LIN {X -289.657,Y 14.097,Z 88.630,A -2.786,B 90.000,C 0.000} C_DIS
LIN {X -289.655,Y 14.148,Z 88.567,A -2.796,B 90.000,C 0.000} C_DIS
LIN {X -289.652,Y 14.199,Z 88.524,A -2.806,B 90.000,C 0.000} C_DIS
LIN {X -289.650,Y 14.241,Z 88.320,A -2.815,B 90.000,C 0.000} C_DIS
LIN {X -289.648,Y 14.292,Z 88.278,A -2.825,B 90.000,C 0.000} C_DIS
LIN {X -289.645,Y 14.343,Z 88.214,A -2.835,B 90.000,C 0.000} C_DIS
LIN {X -289.643,Y 14.385,Z 87.908,A -2.843,B 90.000,C 0.000} C_DIS
LIN {X -289.640,Y 14.436,Z 87.844,A -2.853,B 90.000,C 0.000} C_DIS
LIN {X -289.638,Y 14.487,Z 87.801,A -2.863,B 90.000,C 0.000} C_DIS
LIN {X -289.636,Y 14.530,Z 87.597,A -2.872,B 90.000,C 0.000} C_DIS
LIN {X -289.633,Y 14.581,Z 87.555,A -2.882,B 90.000,C 0.000} C_DIS
LIN {X -289.631,Y 14.632,Z 87.491,A -2.892,B 90.000,C 0.000} C_DIS
LIN {X -289.629,Y 14.674,Z 87.185,A -2.900,B 90.000,C 0.000} C_DIS
LIN {X -289.626,Y 14.725,Z 87.121,A -2.910,B 90.000,C 0.000} C_DIS
LIN {X -289.623,Y 14.776,Z 87.079,A -2.921,B 90.000,C 0.000} C_DIS
LIN {X -289.621,Y 14.818,Z 86.875,A -2.929,B 90.000,C 0.000} C_DIS
LIN {X -289.619,Y 14.869,Z 86.832,A -2.939,B 90.000,C 0.000} C_DIS
LIN {X -289.616,Y 14.920,Z 86.769,A -2.949,B 90.000,C 0.000} C_DIS
LIN {X -289.614,Y 14.963,Z 86.462,A -2.958,B 90.000,C 0.000} C_DIS
LIN {X -289.611,Y 15.014,Z 86.399,A -2.968,B 90.000,C 0.000} C_DIS
LIN {X -289.608,Y 15.065,Z 86.356,A -2.978,B 90.000,C 0.000} C_DIS
LIN {X -289.606,Y 15.107,Z 86.152,A -2.986,B 90.000,C 0.000} C_DIS
LIN {X -289.604,Y 15.158,Z 86.110,A -2.996,B 90.000,C 0.000} C_DIS
LIN {X -289.601,Y 15.209,Z 86.046,A -3.006,B 90.000,C 0.000} C_DIS
LIN {X -289.599,Y 15.251,Z 85.740,A -3.015,B 90.000,C 0.000} C_DIS
LIN {X -289.596,Y 15.302,Z 85.676,A -3.025,B 90.000,C 0.000} C_DIS
LIN {X -289.593,Y 15.353,Z 85.634,A -3.035,B 90.000,C 0.000} C_DIS
LIN {X -289.591,Y 15.396,Z 85.429,A -3.043,B 90.000,C 0.000} C_DIS
LIN {X -289.588,Y 15.447,Z 85.387,A -3.053,B 90.000,C 0.000} C_DIS
LIN {X -289.586,Y 15.498,Z 85.323,A -3.063,B 90.000,C 0.000} C_DIS
LIN {X -289.583,Y 15.540,Z 85.017,A -3.072,B 90.000,C 0.000} C_DIS
LIN {X -289.578,Y 15.642,Z 84.890,A -3.092,B 90.000,C 0.000} C_DIS
LIN {X -289.576,Y 15.684,Z 84.583,A -3.100,B 90.000,C 0.000} C_DIS
LIN {X -289.573,Y 15.735,Z 84.520,A -3.110,B 90.000,C 0.000} C_DIS
LIN {X -289.570,Y 15.786,Z 84.477,A -3.120,B 90.000,C 0.000} C_DIS
LIN {X -289.568,Y 15.829,Z 84.273,A -3.129,B 90.000,C 0.000} C_DIS
LIN {X -289.565,Y 15.880,Z 84.231,A -3.139,B 90.000,C 0.000} C_DIS
LIN {X -289.562,Y 15.931,Z 84.167,A -3.149,B 90.000,C 0.000} C_DIS
LIN {X -289.560,Y 15.973,Z 83.861,A -3.157,B 90.000,C 0.000} C_DIS
LIN {X -289.557,Y 16.024,Z 83.797,A -3.167,B 90.000,C 0.000} C_DIS
LIN {X -289.554,Y 16.075,Z 83.755,A -3.178,B 90.000,C 0.000} C_DIS
LIN {X -289.552,Y 16.117,Z 83.551,A -3.186,B 90.000,C 0.000} C_DIS
LIN {X -289.549,Y 16.168,Z 83.508,A -3.196,B 90.000,C 0.000} C_DIS
LIN {X -289.546,Y 16.219,Z 83.444,A -3.206,B 90.000,C 0.000} C_DIS
LIN {X -289.544,Y 16.262,Z 83.138,A -3.214,B 90.000,C 0.000} C_DIS
LIN {X -289.541,Y 16.312,Z 83.075,A -3.225,B 90.000,C 0.000} C_DIS
LIN {X -289.538,Y 16.363,Z 83.032,A -3.235,B 90.000,C 0.000} C_DIS
LIN {X -289.536,Y 16.406,Z 82.828,A -3.243,B 90.000,C 0.000} C_DIS
LIN {X -289.533,Y 16.457,Z 82.785,A -3.253,B 90.000,C 0.000} C_DIS
LIN {X -289.530,Y 16.508,Z 82.722,A -3.263,B 90.000,C 0.000} C_DIS
LIN {X -289.527,Y 16.550,Z 82.416,A -3.272,B 90.000,C 0.000} C_DIS
LIN {X -289.524,Y 16.601,Z 82.352,A -3.282,B 90.000,C 0.000} C_DIS
LIN {X -289.522,Y 16.652,Z 82.309,A -3.292,B 90.000,C 0.000} C_DIS
LIN {X -289.519,Y 16.694,Z 82.105,A -3.300,B 90.000,C 0.000} C_DIS
LIN {X -289.516,Y 16.745,Z 82.063,A -3.310,B 90.000,C 0.000} C_DIS
LIN {X -289.513,Y 16.796,Z 81.999,A -3.320,B 90.000,C 0.000} C_DIS
LIN {X -289.511,Y 16.839,Z 81.693,A -3.329,B 90.000,C 0.000} C_DIS
LIN {X -289.508,Y 16.890,Z 81.629,A -3.339,B 90.000,C 0.000} C_DIS
LIN {X -289.505,Y 16.941,Z 81.587,A -3.349,B 90.000,C 0.000} C_DIS
LIN {X -289.502,Y 16.983,Z 81.383,A -3.357,B 90.000,C 0.000} C_DIS
LIN {X -289.499,Y 17.034,Z 81.340,A -3.367,B 90.000,C 0.000} C_DIS
LIN {X -289.496,Y 17.085,Z 81.276,A -3.377,B 90.000,C 0.000} C_DIS
LIN {X -289.494,Y 17.127,Z 80.970,A -3.386,B 90.000,C 0.000} C_DIS
LIN {X -289.491,Y 17.178,Z 80.907,A -3.396,B 90.000,C 0.000} C_DIS
LIN {X -289.488,Y 17.229,Z 80.864,A -3.406,B 90.000,C 0.000} C_DIS
LIN {X -289.485,Y 17.272,Z 80.660,A -3.414,B 90.000,C 0.000} C_DIS
LIN {X -289.482,Y 17.322,Z 80.618,A -3.424,B 90.000,C 0.000} C_DIS
LIN {X -289.479,Y 17.373,Z 80.554,A -3.435,B 90.000,C 0.000} C_DIS
LIN {X -289.477,Y 17.416,Z 80.248,A -3.443,B 90.000,C 0.000} C_DIS
LIN {X -289.474,Y 17.467,Z 80.184,A -3.453,B 90.000,C 0.000} C_DIS
LIN {X -289.470,Y 17.518,Z 80.141,A -3.463,B 90.000,C 0.000} C_DIS
LIN {X -289.468,Y 17.560,Z 79.937,A -3.471,B 90.000,C 0.000} C_DIS
LIN {X -289.465,Y 17.611,Z 79.895,A -3.482,B 90.000,C 0.000} C_DIS
LIN {X -289.462,Y 17.662,Z 79.831,A -3.492,B 90.000,C 0.000} C_DIS
LIN {X -289.459,Y 17.704,Z 79.525,A -3.500,B 90.000,C 0.000} C_DIS
LIN {X -289.456,Y 17.755,Z 79.461,A -3.510,B 90.000,C 0.000} C_DIS
LIN {X -289.453,Y 17.806,Z 79.419,A -3.520,B 90.000,C 0.000} C_DIS
LIN {X -289.450,Y 17.849,Z 79.215,A -3.529,B 90.000,C 0.000} C_DIS
LIN {X -289.447,Y 17.900,Z 79.172,A -3.539,B 90.000,C 0.000} C_DIS
LIN {X -289.444,Y 17.950,Z 79.109,A -3.549,B 90.000,C 0.000} C_DIS
LIN {X -289.441,Y 17.993,Z 78.802,A -3.557,B 90.000,C 0.000} C_DIS
LIN {X -289.438,Y 18.044,Z 78.739,A -3.567,B 90.000,C 0.000} C_DIS
LIN {X -289.435,Y 18.095,Z 78.696,A -3.577,B 90.000,C 0.000} C_DIS
LIN {X -289.432,Y 18.137,Z 78.492,A -3.586,B 90.000,C 0.000} C_DIS
LIN {X -289.429,Y 18.188,Z 78.450,A -3.596,B 90.000,C 0.000} C_DIS
LIN {X -289.426,Y 18.239,Z 78.386,A -3.606,B 90.000,C 0.000} C_DIS
LIN {X -289.423,Y 18.281,Z 78.080,A -3.614,B 90.000,C 0.000} C_DIS
LIN {X -289.420,Y 18.332,Z 78.016,A -3.624,B 90.000,C 0.000} C_DIS
LIN {X -289.417,Y 18.383,Z 77.974,A -3.634,B 90.000,C 0.000} C_DIS
LIN {X -289.414,Y 18.426,Z 77.769,A -3.643,B 90.000,C 0.000} C_DIS
LIN {X -289.411,Y 18.476,Z 77.727,A -3.653,B 90.000,C 0.000} C_DIS
LIN {X -289.408,Y 18.527,Z 77.663,A -3.663,B 90.000,C 0.000} C_DIS
LIN {X -289.405,Y 18.570,Z 77.357,A -3.671,B 90.000,C 0.000} C_DIS
LIN {X -289.402,Y 18.621,Z 77.293,A -3.681,B 90.000,C 0.000} C_DIS
LIN {X -289.398,Y 18.672,Z 77.251,A -3.692,B 90.000,C 0.000} C_DIS
LIN {X -289.396,Y 18.714,Z 77.047,A -3.700,B 90.000,C 0.000} C_DIS
LIN {X -289.392,Y 18.765,Z 77.004,A -3.710,B 90.000,C 0.000} C_DIS
LIN {X -289.389,Y 18.816,Z 76.941,A -3.720,B 90.000,C 0.000} C_DIS
LIN {X -289.386,Y 18.858,Z 76.634,A -3.728,B 90.000,C 0.000} C_DIS
LIN {X -289.383,Y 18.909,Z 76.571,A -3.739,B 90.000,C 0.000} C_DIS
LIN {X -289.380,Y 18.960,Z 76.528,A -3.749,B 90.000,C 0.000} C_DIS
LIN {X -289.377,Y 19.002,Z 76.324,A -3.757,B 90.000,C 0.000} C_DIS
LIN {X -289.373,Y 19.053,Z 76.282,A -3.767,B 90.000,C 0.000} C_DIS
LIN {X -289.370,Y 19.104,Z 76.218,A -3.777,B 90.000,C 0.000} C_DIS
LIN {X -289.367,Y 19.147,Z 75.912,A -3.786,B 90.000,C 0.000} C_DIS
LIN {X -289.364,Y 19.198,Z 75.848,A -3.796,B 90.000,C 0.000} C_DIS
LIN {X -289.360,Y 19.249,Z 75.806,A -3.806,B 90.000,C 0.000} C_DIS
LIN {X -289.358,Y 19.291,Z 75.601,A -3.814,B 90.000,C 0.000} C_DIS
LIN {X -289.354,Y 19.342,Z 75.559,A -3.824,B 90.000,C 0.000} C_DIS
LIN {X -289.351,Y 19.393,Z 75.495,A -3.834,B 90.000,C 0.000} C_DIS
LIN {X -289.348,Y 19.435,Z 75.189,A -3.843,B 90.000,C 0.000} C_DIS
LIN {X -289.345,Y 19.486,Z 75.125,A -3.853,B 90.000,C 0.000} C_DIS
LIN {X -289.341,Y 19.537,Z 75.083,A -3.863,B 90.000,C 0.000} C_DIS
LIN {X -289.338,Y 19.579,Z 74.879,A -3.871,B 90.000,C 0.000} C_DIS
LIN {X -289.335,Y 19.630,Z 74.836,A -3.881,B 90.000,C 0.000} C_DIS
LIN {X -289.331,Y 19.681,Z 74.773,A -3.891,B 90.000,C 0.000} C_DIS
LIN {X -289.329,Y 19.723,Z 74.466,A -3.900,B 90.000,C 0.000} C_DIS
LIN {X -289.325,Y 19.774,Z 74.403,A -3.910,B 90.000,C 0.000} C_DIS
LIN {X -289.322,Y 19.825,Z 74.360,A -3.920,B 90.000,C 0.000} C_DIS
LIN {X -289.319,Y 19.868,Z 74.156,A -3.928,B 90.000,C 0.000} C_DIS
LIN {X -289.315,Y 19.919,Z 74.114,A -3.938,B 90.000,C 0.000} C_DIS
LIN {X -289.312,Y 19.970,Z 74.050,A -3.949,B 90.000,C 0.000} C_DIS
LIN {X -289.309,Y 20.012,Z 73.744,A -3.957,B 90.000,C 0.000} C_DIS
LIN {X -289.305,Y 20.063,Z 73.680,A -3.967,B 90.000,C 0.000} C_DIS
LIN {X -289.302,Y 20.114,Z 73.638,A -3.977,B 90.000,C 0.000} C_DIS
LIN {X -289.299,Y 20.156,Z 73.434,A -3.985,B 90.000,C 0.000} C_DIS
LIN {X -289.295,Y 20.207,Z 73.391,A -3.996,B 90.000,C 0.000} C_DIS
LIN {X -289.292,Y 20.258,Z 73.327,A -4.006,B 90.000,C 0.000} C_DIS
LIN {X -289.289,Y 20.300,Z 73.021,A -4.014,B 90.000,C 0.000} C_DIS
LIN {X -289.281,Y 20.402,Z 72.894,A -4.034,B 90.000,C 0.000} C_DIS
LIN {X -289.278,Y 20.444,Z 72.588,A -4.043,B 90.000,C 0.000} C_DIS
LIN {X -289.275,Y 20.495,Z 72.524,A -4.053,B 90.000,C 0.000} C_DIS
LIN {X -289.271,Y 20.546,Z 72.481,A -4.063,B 90.000,C 0.000} C_DIS
LIN {X -289.268,Y 20.589,Z 72.277,A -4.071,B 90.000,C 0.000} C_DIS
LIN {X -289.265,Y 20.639,Z 72.235,A -4.081,B 90.000,C 0.000} C_DIS
LIN {X -289.261,Y 20.690,Z 72.171,A -4.091,B 90.000,C 0.000} C_DIS
LIN {X -289.258,Y 20.733,Z 71.865,A -4.100,B 90.000,C 0.000} C_DIS
LIN {X -289.254,Y 20.784,Z 71.801,A -4.110,B 90.000,C 0.000} C_DIS
LIN {X -289.251,Y 20.835,Z 71.759,A -4.120,B 90.000,C 0.000} C_DIS
LIN {X -289.248,Y 20.877,Z 71.555,A -4.128,B 90.000,C 0.000} C_DIS
LIN {X -289.244,Y 20.928,Z 71.512,A -4.138,B 90.000,C 0.000} C_DIS
LIN {X -289.240,Y 20.979,Z 71.449,A -4.148,B 90.000,C 0.000} C_DIS
LIN {X -289.237,Y 21.021,Z 71.142,A -4.157,B 90.000,C 0.000} C_DIS
LIN {X -289.233,Y 21.072,Z 71.079,A -4.167,B 90.000,C 0.000} C_DIS
LIN {X -289.230,Y 21.123,Z 71.036,A -4.177,B 90.000,C 0.000} C_DIS
LIN {X -289.227,Y 21.165,Z 70.832,A -4.185,B 90.000,C 0.000} C_DIS
LIN {X -289.223,Y 21.216,Z 70.790,A -4.195,B 90.000,C 0.000} C_DIS
LIN {X -289.219,Y 21.267,Z 70.726,A -4.206,B 90.000,C 0.000} C_DIS
LIN {X -289.216,Y 21.309,Z 70.420,A -4.214,B 90.000,C 0.000} C_DIS
LIN {X -289.212,Y 21.360,Z 70.356,A -4.224,B 90.000,C 0.000} C_DIS
LIN {X -289.209,Y 21.411,Z 70.314,A -4.234,B 90.000,C 0.000} C_DIS
LIN {X -289.205,Y 21.453,Z 70.109,A -4.242,B 90.000,C 0.000} C_DIS
LIN {X -289.202,Y 21.504,Z 70.067,A -4.253,B 90.000,C 0.000} C_DIS
LIN {X -289.198,Y 21.555,Z 70.003,A -4.263,B 90.000,C 0.000} C_DIS
LIN {X -289.195,Y 21.598,Z 69.697,A -4.271,B 90.000,C 0.000} C_DIS
LIN {X -289.191,Y 21.648,Z 69.633,A -4.281,B 90.000,C 0.000} C_DIS
LIN {X -289.187,Y 21.699,Z 69.591,A -4.291,B 90.000,C 0.000} C_DIS
LIN {X -289.184,Y 21.742,Z 69.387,A -4.300,B 90.000,C 0.000} C_DIS
LIN {X -289.180,Y 21.793,Z 69.344,A -4.310,B 90.000,C 0.000} C_DIS
LIN {X -289.176,Y 21.843,Z 69.281,A -4.320,B 90.000,C 0.000} C_DIS
LIN {X -289.173,Y 21.886,Z 68.974,A -4.328,B 90.000,C 0.000} C_DIS
LIN {X -289.169,Y 21.937,Z 68.911,A -4.338,B 90.000,C 0.000} C_DIS
LIN {X -289.165,Y 21.988,Z 68.868,A -4.348,B 90.000,C 0.000} C_DIS
LIN {X -289.162,Y 22.030,Z 68.664,A -4.357,B 90.000,C 0.000} C_DIS
LIN {X -289.158,Y 22.081,Z 68.622,A -4.367,B 90.000,C 0.000} C_DIS
LIN {X -289.154,Y 22.132,Z 68.558,A -4.377,B 90.000,C 0.000} C_DIS
LIN {X -289.151,Y 22.174,Z 68.252,A -4.385,B 90.000,C 0.000} C_DIS
LIN {X -289.147,Y 22.225,Z 68.188,A -4.395,B 90.000,C 0.000} C_DIS
LIN {X -289.143,Y 22.276,Z 68.146,A -4.405,B 90.000,C 0.000} C_DIS
LIN {X -289.140,Y 22.318,Z 67.941,A -4.414,B 90.000,C 0.000} C_DIS
LIN {X -289.136,Y 22.369,Z 67.899,A -4.424,B 90.000,C 0.000} C_DIS
LIN {X -289.132,Y 22.420,Z 67.835,A -4.434,B 90.000,C 0.000} C_DIS
LIN {X -289.129,Y 22.462,Z 67.529,A -4.442,B 90.000,C 0.000} C_DIS
LIN {X -289.125,Y 22.513,Z 67.465,A -4.452,B 90.000,C 0.000} C_DIS
LIN {X -289.121,Y 22.564,Z 67.423,A -4.463,B 90.000,C 0.000} C_DIS
LIN {X -289.118,Y 22.606,Z 67.219,A -4.471,B 90.000,C 0.000} C_DIS
LIN {X -289.114,Y 22.657,Z 67.176,A -4.481,B 90.000,C 0.000} C_DIS
LIN {X -289.110,Y 22.708,Z 67.113,A -4.491,B 90.000,C 0.000} C_DIS
LIN {X -289.106,Y 22.750,Z 66.806,A -4.499,B 90.000,C 0.000} C_DIS
LIN {X -289.102,Y 22.801,Z 66.743,A -4.510,B 90.000,C 0.000} C_DIS
LIN {X -289.098,Y 22.852,Z 66.700,A -4.520,B 90.000,C 0.000} C_DIS
LIN {X -289.095,Y 22.894,Z 66.496,A -4.528,B 90.000,C 0.000} C_DIS
LIN {X -289.091,Y 22.945,Z 66.454,A -4.538,B 90.000,C 0.000} C_DIS
LIN {X -289.087,Y 22.996,Z 66.390,A -4.548,B 90.000,C 0.000} C_DIS
LIN {X -289.083,Y 23.039,Z 66.084,A -4.557,B 90.000,C 0.000} C_DIS
LIN {X -289.079,Y 23.089,Z 66.020,A -4.567,B 90.000,C 0.000} C_DIS
LIN {X -289.075,Y 23.140,Z 65.978,A -4.577,B 90.000,C 0.000} C_DIS
LIN {X -289.072,Y 23.183,Z 65.774,A -4.585,B 90.000,C 0.000} C_DIS
LIN {X -289.068,Y 23.234,Z 65.731,A -4.595,B 90.000,C 0.000} C_DIS
LIN {X -289.064,Y 23.284,Z 65.667,A -4.605,B 90.000,C 0.000} C_DIS
LIN {X -289.060,Y 23.327,Z 65.361,A -4.614,B 90.000,C 0.000} C_DIS
LIN {X -289.056,Y 23.378,Z 65.298,A -4.624,B 90.000,C 0.000} C_DIS
LIN {X -289.052,Y 23.428,Z 65.255,A -4.634,B 90.000,C 0.000} C_DIS
LIN {X -289.049,Y 23.471,Z 65.051,A -4.642,B 90.000,C 0.000} C_DIS
LIN {X -289.045,Y 23.522,Z 65.008,A -4.652,B 90.000,C 0.000} C_DIS
LIN {X -289.040,Y 23.572,Z 64.945,A -4.662,B 90.000,C 0.000} C_DIS
LIN {X -289.037,Y 23.615,Z 64.639,A -4.671,B 90.000,C 0.000} C_DIS
LIN {X -289.033,Y 23.666,Z 64.575,A -4.681,B 90.000,C 0.000} C_DIS
LIN {X -289.029,Y 23.717,Z 64.532,A -4.691,B 90.000,C 0.000} C_DIS
LIN {X -289.025,Y 23.759,Z 64.328,A -4.699,B 90.000,C 0.000} C_DIS
LIN {X -289.021,Y 23.810,Z 64.286,A -4.709,B 90.000,C 0.000} C_DIS
LIN {X -289.017,Y 23.861,Z 64.222,A -4.720,B 90.000,C 0.000} C_DIS
LIN {X -289.013,Y 23.903,Z 63.916,A -4.728,B 90.000,C 0.000} C_DIS
LIN {X -289.009,Y 23.954,Z 63.852,A -4.738,B 90.000,C 0.000} C_DIS
LIN {X -289.005,Y 24.005,Z 63.810,A -4.748,B 90.000,C 0.000} C_DIS
LIN {X -289.001,Y 24.047,Z 63.606,A -4.756,B 90.000,C 0.000} C_DIS
LIN {X -288.997,Y 24.098,Z 63.563,A -4.767,B 90.000,C 0.000} C_DIS
LIN {X -288.993,Y 24.149,Z 63.500,A -4.777,B 90.000,C 0.000} C_DIS
LIN {X -288.989,Y 24.191,Z 63.193,A -4.785,B 90.000,C 0.000} C_DIS
LIN {X -288.985,Y 24.242,Z 63.130,A -4.795,B 90.000,C 0.000} C_DIS
LIN {X -288.981,Y 24.293,Z 63.087,A -4.805,B 90.000,C 0.000} C_DIS
LIN {X -288.977,Y 24.335,Z 62.883,A -4.814,B 90.000,C 0.000} C_DIS
LIN {X -288.973,Y 24.386,Z 62.841,A -4.824,B 90.000,C 0.000} C_DIS
LIN {X -288.969,Y 24.437,Z 62.777,A -4.834,B 90.000,C 0.000} C_DIS
LIN {X -288.965,Y 24.479,Z 62.471,A -4.842,B 90.000,C 0.000} C_DIS
LIN {X -288.961,Y 24.530,Z 62.407,A -4.852,B 90.000,C 0.000} C_DIS
LIN {X -288.956,Y 24.581,Z 62.365,A -4.862,B 90.000,C 0.000} C_DIS
LIN {X -288.953,Y 24.623,Z 62.160,A -4.871,B 90.000,C 0.000} C_DIS
LIN {X -288.948,Y 24.674,Z 62.118,A -4.881,B 90.000,C 0.000} C_DIS
LIN {X -288.944,Y 24.725,Z 62.054,A -4.891,B 90.000,C 0.000} C_DIS
LIN {X -288.940,Y 24.767,Z 61.748,A -4.899,B 90.000,C 0.000} C_DIS
LIN {X -288.936,Y 24.818,Z 61.684,A -4.909,B 90.000,C 0.000} C_DIS
LIN {X -288.932,Y 24.869,Z 61.642,A -4.919,B 90.000,C 0.000} C_DIS
LIN {X -288.928,Y 24.911,Z 61.438,A -4.928,B 90.000,C 0.000} C_DIS
LIN {X -288.924,Y 24.962,Z 61.395,A -4.938,B 90.000,C 0.000} C_DIS
LIN {X -288.919,Y 25.013,Z 61.332,A -4.948,B 90.000,C 0.000} C_DIS
LIN {X -288.916,Y 25.055,Z 61.025,A -4.956,B 90.000,C 0.000} C_DIS
LIN {X -288.911,Y 25.106,Z 60.962,A -4.966,B 90.000,C 0.000} C_DIS
LIN {X -288.907,Y 25.157,Z 60.919,A -4.977,B 90.000,C 0.000} C_DIS
LIN {X -288.903,Y 25.199,Z 60.715,A -4.985,B 90.000,C 0.000} C_DIS
LIN {X -288.899,Y 25.250,Z 60.673,A -4.995,B 90.000,C 0.000} C_DIS
LIN {X -288.894,Y 25.301,Z 60.609,A -5.005,B 90.000,C 0.000} C_DIS
LIN {X -288.891,Y 25.343,Z 60.303,A -5.013,B 90.000,C 0.000} C_DIS
LIN {X -288.882,Y 25.445,Z 60.175,A -5.034,B 90.000,C 0.000} C_DIS
LIN {X -288.878,Y 25.487,Z 59.869,A -5.042,B 90.000,C 0.000} C_DIS
LIN {X -288.873,Y 25.538,Z 59.805,A -5.052,B 90.000,C 0.000} C_DIS
LIN {X -288.869,Y 25.589,Z 59.763,A -5.062,B 90.000,C 0.000} C_DIS
LIN {X -288.865,Y 25.631,Z 59.559,A -5.071,B 90.000,C 0.000} C_DIS
LIN {X -288.861,Y 25.682,Z 59.516,A -5.081,B 90.000,C 0.000} C_DIS
LIN {X -288.856,Y 25.733,Z 59.453,A -5.091,B 90.000,C 0.000} C_DIS
LIN {X -288.852,Y 25.775,Z 59.146,A -5.099,B 90.000,C 0.000} C_DIS
LIN {X -288.848,Y 25.826,Z 59.083,A -5.109,B 90.000,C 0.000} C_DIS
LIN {X -288.843,Y 25.877,Z 59.040,A -5.119,B 90.000,C 0.000} C_DIS
LIN {X -288.839,Y 25.919,Z 58.836,A -5.128,B 90.000,C 0.000} C_DIS
LIN {X -288.835,Y 25.970,Z 58.794,A -5.138,B 90.000,C 0.000} C_DIS
LIN {X -288.830,Y 26.020,Z 58.730,A -5.148,B 90.000,C 0.000} C_DIS
LIN {X -288.826,Y 26.063,Z 58.424,A -5.156,B 90.000,C 0.000} C_DIS
LIN {X -288.822,Y 26.114,Z 58.360,A -5.166,B 90.000,C 0.000} C_DIS
LIN {X -288.817,Y 26.164,Z 58.318,A -5.176,B 90.000,C 0.000} C_DIS
LIN {X -288.813,Y 26.207,Z 58.114,A -5.185,B 90.000,C 0.000} C_DIS
LIN {X -288.809,Y 26.258,Z 58.071,A -5.195,B 90.000,C 0.000} C_DIS
LIN {X -288.804,Y 26.308,Z 58.007,A -5.205,B 90.000,C 0.000} C_DIS
LIN {X -288.800,Y 26.351,Z 57.701,A -5.213,B 90.000,C 0.000} C_DIS
LIN {X -288.796,Y 26.401,Z 57.638,A -5.223,B 90.000,C 0.000} C_DIS
LIN {X -288.791,Y 26.452,Z 57.595,A -5.233,B 90.000,C 0.000} C_DIS
LIN {X -288.787,Y 26.495,Z 57.391,A -5.242,B 90.000,C 0.000} C_DIS
LIN {X -288.783,Y 26.545,Z 57.348,A -5.252,B 90.000,C 0.000} C_DIS
LIN {X -288.778,Y 26.596,Z 57.285,A -5.262,B 90.000,C 0.000} C_DIS
LIN {X -288.774,Y 26.638,Z 56.979,A -5.270,B 90.000,C 0.000} C_DIS
LIN {X -288.769,Y 26.689,Z 56.915,A -5.281,B 90.000,C 0.000} C_DIS
LIN {X -288.765,Y 26.740,Z 56.872,A -5.291,B 90.000,C 0.000} C_DIS
LIN {X -288.761,Y 26.782,Z 56.668,A -5.299,B 90.000,C 0.000} C_DIS
LIN {X -288.756,Y 26.833,Z 56.626,A -5.309,B 90.000,C 0.000} C_DIS
LIN {X -288.751,Y 26.884,Z 56.562,A -5.319,B 90.000,C 0.000} C_DIS
LIN {X -288.747,Y 26.926,Z 56.256,A -5.328,B 90.000,C 0.000} C_DIS
LIN {X -288.743,Y 26.977,Z 56.192,A -5.338,B 90.000,C 0.000} C_DIS
LIN {X -288.738,Y 27.028,Z 56.150,A -5.348,B 90.000,C 0.000} C_DIS
LIN {X -288.734,Y 27.070,Z 55.946,A -5.356,B 90.000,C 0.000} C_DIS
LIN {X -288.729,Y 27.121,Z 55.903,A -5.366,B 90.000,C 0.000} C_DIS
LIN {X -288.724,Y 27.172,Z 55.840,A -5.376,B 90.000,C 0.000} C_DIS
LIN {X -288.720,Y 27.214,Z 55.533,A -5.385,B 90.000,C 0.000} C_DIS
LIN {X -288.715,Y 27.265,Z 55.470,A -5.395,B 90.000,C 0.000} C_DIS
LIN {X -288.711,Y 27.316,Z 55.427,A -5.405,B 90.000,C 0.000} C_DIS
LIN {X -288.707,Y 27.358,Z 55.223,A -5.413,B 90.000,C 0.000} C_DIS
LIN {X -288.702,Y 27.409,Z 55.181,A -5.423,B 90.000,C 0.000} C_DIS
LIN {X -288.697,Y 27.460,Z 55.117,A -5.433,B 90.000,C 0.000} C_DIS
LIN {X -288.693,Y 27.502,Z 54.811,A -5.442,B 90.000,C 0.000} C_DIS
LIN {X -288.688,Y 27.553,Z 54.747,A -5.452,B 90.000,C 0.000} C_DIS
LIN {X -288.683,Y 27.603,Z 54.705,A -5.462,B 90.000,C 0.000} C_DIS
LIN {X -288.679,Y 27.646,Z 54.500,A -5.470,B 90.000,C 0.000} C_DIS
LIN {X -288.674,Y 27.697,Z 54.458,A -5.480,B 90.000,C 0.000} C_DIS
LIN {X -288.670,Y 27.747,Z 54.394,A -5.490,B 90.000,C 0.000} C_DIS
LIN {X -288.665,Y 27.790,Z 54.088,A -5.499,B 90.000,C 0.000} C_DIS
LIN {X -288.661,Y 27.840,Z 54.024,A -5.509,B 90.000,C 0.000} C_DIS
LIN {X -288.656,Y 27.891,Z 53.982,A -5.519,B 90.000,C 0.000} C_DIS
LIN {X -288.652,Y 27.933,Z 53.778,A -5.527,B 90.000,C 0.000} C_DIS
LIN {X -288.647,Y 27.984,Z 53.735,A -5.538,B 90.000,C 0.000} C_DIS
LIN {X -288.642,Y 28.035,Z 53.672,A -5.548,B 90.000,C 0.000} C_DIS
LIN {X -288.638,Y 28.077,Z 53.365,A -5.556,B 90.000,C 0.000} C_DIS
LIN {X -288.633,Y 28.128,Z 53.302,A -5.566,B 90.000,C 0.000} C_DIS
LIN {X -288.628,Y 28.179,Z 53.259,A -5.576,B 90.000,C 0.000} C_DIS
LIN {X -288.624,Y 28.221,Z 53.055,A -5.585,B 90.000,C 0.000} C_DIS
LIN {X -288.619,Y 28.272,Z 53.013,A -5.595,B 90.000,C 0.000} C_DIS
LIN {X -288.614,Y 28.323,Z 52.949,A -5.605,B 90.000,C 0.000} C_DIS
LIN {X -288.609,Y 28.365,Z 52.643,A -5.613,B 90.000,C 0.000} C_DIS
LIN {X -288.604,Y 28.416,Z 52.579,A -5.623,B 90.000,C 0.000} C_DIS
LIN {X -288.599,Y 28.467,Z 52.537,A -5.633,B 90.000,C 0.000} C_DIS
LIN {X -288.595,Y 28.509,Z 52.332,A -5.642,B 90.000,C 0.000} C_DIS
LIN {X -288.590,Y 28.560,Z 52.290,A -5.652,B 90.000,C 0.000} C_DIS
LIN {X -288.585,Y 28.610,Z 52.226,A -5.662,B 90.000,C 0.000} C_DIS
LIN {X -288.581,Y 28.653,Z 51.920,A -5.670,B 90.000,C 0.000} C_DIS
LIN {X -288.576,Y 28.703,Z 51.856,A -5.680,B 90.000,C 0.000} C_DIS
LIN {X -288.571,Y 28.754,Z 51.814,A -5.690,B 90.000,C 0.000} C_DIS
LIN {X -288.567,Y 28.796,Z 51.610,A -5.699,B 90.000,C 0.000} C_DIS
LIN {X -288.562,Y 28.847,Z 51.567,A -5.709,B 90.000,C 0.000} C_DIS
LIN {X -288.557,Y 28.898,Z 51.504,A -5.719,B 90.000,C 0.000} C_DIS
LIN {X -288.552,Y 28.940,Z 51.197,A -5.727,B 90.000,C 0.000} C_DIS
LIN {X -288.547,Y 28.991,Z 51.134,A -5.737,B 90.000,C 0.000} C_DIS
LIN {X -288.542,Y 29.042,Z 51.091,A -5.747,B 90.000,C 0.000} C_DIS
LIN {X -288.538,Y 29.084,Z 50.887,A -5.756,B 90.000,C 0.000} C_DIS
LIN {X -288.533,Y 29.135,Z 50.845,A -5.766,B 90.000,C 0.000} C_DIS
LIN {X -288.528,Y 29.186,Z 50.781,A -5.776,B 90.000,C 0.000} C_DIS
LIN {X -288.523,Y 29.228,Z 50.475,A -5.784,B 90.000,C 0.000} C_DIS
LIN {X -288.518,Y 29.279,Z 50.411,A -5.795,B 90.000,C 0.000} C_DIS
LIN {X -288.513,Y 29.329,Z 50.369,A -5.805,B 90.000,C 0.000} C_DIS
LIN {X -288.509,Y 29.372,Z 50.165,A -5.813,B 90.000,C 0.000} C_DIS
LIN {X -288.504,Y 29.422,Z 50.122,A -5.823,B 90.000,C 0.000} C_DIS
LIN {X -288.498,Y 29.473,Z 50.058,A -5.833,B 90.000,C 0.000} C_DIS
LIN {X -288.494,Y 29.515,Z 49.752,A -5.842,B 90.000,C 0.000} C_DIS
LIN {X -288.489,Y 29.566,Z 49.688,A -5.852,B 90.000,C 0.000} C_DIS
LIN {X -288.484,Y 29.617,Z 49.646,A -5.862,B 90.000,C 0.000} C_DIS
LIN {X -288.479,Y 29.659,Z 49.442,A -5.870,B 90.000,C 0.000} C_DIS
LIN {X -288.474,Y 29.710,Z 49.399,A -5.880,B 90.000,C 0.000} C_DIS
LIN {X -288.469,Y 29.761,Z 49.336,A -5.890,B 90.000,C 0.000} C_DIS
LIN {X -288.465,Y 29.803,Z 49.030,A -5.899,B 90.000,C 0.000} C_DIS
LIN {X -288.459,Y 29.854,Z 48.966,A -5.909,B 90.000,C 0.000} C_DIS
LIN {X -288.454,Y 29.905,Z 48.923,A -5.919,B 90.000,C 0.000} C_DIS
LIN {X -288.450,Y 29.947,Z 48.719,A -5.927,B 90.000,C 0.000} C_DIS
LIN {X -288.444,Y 29.998,Z 48.677,A -5.937,B 90.000,C 0.000} C_DIS
LIN {X -288.439,Y 30.048,Z 48.613,A -5.947,B 90.000,C 0.000} C_DIS
LIN {X -288.435,Y 30.091,Z 48.307,A -5.956,B 90.000,C 0.000} C_DIS
LIN {X -288.429,Y 30.141,Z 48.243,A -5.966,B 90.000,C 0.000} C_DIS
LIN {X -288.424,Y 30.192,Z 48.201,A -5.976,B 90.000,C 0.000} C_DIS
LIN {X -288.420,Y 30.234,Z 47.997,A -5.984,B 90.000,C 0.000} C_DIS
LIN {X -288.414,Y 30.285,Z 47.954,A -5.994,B 90.000,C 0.000} C_DIS
LIN {X -288.409,Y 30.336,Z 47.890,A -6.004,B 90.000,C 0.000} C_DIS
LIN {X -288.405,Y 30.378,Z 47.584,A -6.013,B 90.000,C 0.000} C_DIS
LIN {X -288.394,Y 30.480,Z 47.457,A -6.033,B 90.000,C 0.000} C_DIS
LIN {X -288.389,Y 30.522,Z 47.151,A -6.041,B 90.000,C 0.000} C_DIS
LIN {X -288.384,Y 30.572,Z 47.087,A -6.051,B 90.000,C 0.000} C_DIS
LIN {X -288.379,Y 30.623,Z 47.045,A -6.062,B 90.000,C 0.000} C_DIS
LIN {X -288.374,Y 30.665,Z 46.840,A -6.070,B 90.000,C 0.000} C_DIS
LIN {X -288.363,Y 30.767,Z 46.755,A -6.090,B 90.000,C 0.000} C_DIS
LIN {X -288.359,Y 30.809,Z 46.551,A -6.099,B 90.000,C 0.000} C_DIS
LIN {X -288.353,Y 30.860,Z 46.509,A -6.109,B 90.000,C 0.000} C_DIS
LIN {X -288.348,Y 30.911,Z 46.450,A -6.119,B 90.000,C 0.000} C_DIS
LIN {X -288.341,Y 30.972,Z 46.134,A -6.131,B 90.000,C 0.000} C_DIS
LIN {X -288.319,Y 31.177,Z 45.892,A -6.172,B 90.000,C 0.000} C_DIS
LIN {X -288.315,Y 31.219,Z 45.770,A -6.180,B 90.000,C 0.000} C_DIS
LIN {X -288.312,Y 31.240,Z 45.679,A -6.184,B 90.000,C 0.000} C_DIS
LIN {X -288.301,Y 31.342,Z 45.604,A -6.204,B 90.000,C 0.000} C_DIS
LIN {X -288.299,Y 31.363,Z 45.513,A -6.209,B 90.000,C 0.000} C_DIS
LIN {X -288.295,Y 31.405,Z 45.392,A -6.217,B 90.000,C 0.000} C_DIS
LIN {X -288.283,Y 31.507,Z 45.280,A -6.237,B 90.000,C 0.000} C_DIS
LIN {X -288.245,Y 31.861,Z 44.803,A -6.307,B 90.000,C 0.000} C_DIS
LIN {X -288.136,Y 32.827,Z 43.830,A -6.500,B 90.000,C 0.000} C_DIS
LIN {X -288.082,Y 33.302,Z 43.474,A -6.594,B 90.000,C 0.000} C_DIS
LIN {X -288.069,Y 33.412,Z 43.372,A -6.616,B 90.000,C 0.000} C_DIS
LIN {X -288.055,Y 33.533,Z 43.329,A -6.640,B 90.000,C 0.000} C_DIS
LIN {X -288.044,Y 33.623,Z 43.308,A -6.658,B 90.000,C 0.000} C_DIS
LIN {X -288.035,Y 33.703,Z 43.206,A -6.674,B 90.000,C 0.000} C_DIS
LIN {X -288.011,Y 33.906,Z 43.163,A -6.714,B 90.000,C 0.000} C_DIS
LIN {X -288.001,Y 33.990,Z 43.061,A -6.731,B 90.000,C 0.000} C_DIS
LIN {X -287.977,Y 34.193,Z 43.019,A -6.771,B 90.000,C 0.000} C_DIS
LIN {X -287.972,Y 34.235,Z 42.968,A -6.780,B 90.000,C 0.000} C_DIS
LIN {X -287.965,Y 34.298,Z 42.917,A -6.792,B 90.000,C 0.000} C_DIS
LIN {X -287.928,Y 34.602,Z 42.874,A -6.853,B 90.000,C 0.000} C_DIS
LIN {X -287.913,Y 34.729,Z 42.772,A -6.878,B 90.000,C 0.000} C_DIS
LIN {X -287.876,Y 35.033,Z 42.730,A -6.938,B 90.000,C 0.000} C_DIS
LIN {X -287.869,Y 35.096,Z 42.679,A -6.951,B 90.000,C 0.000} C_DIS
LIN {X -287.836,Y 35.365,Z 42.626,A -7.005,B 90.000,C 0.000} C_DIS
LIN {X -287.651,Y 36.835,Z 42.626,A -7.297,B 90.000,C 0.000} C_DIS
LIN {X -287.617,Y 37.103,Z 42.679,A -7.351,B 90.000,C 0.000} C_DIS
LIN {X -287.606,Y 37.188,Z 42.730,A -7.368,B 90.000,C 0.000} C_DIS
LIN {X -287.553,Y 37.593,Z 42.772,A -7.448,B 90.000,C 0.000} C_DIS
LIN {X -287.542,Y 37.677,Z 42.823,A -7.465,B 90.000,C 0.000} C_DIS
LIN {X -287.534,Y 37.740,Z 42.874,A -7.478,B 90.000,C 0.000} C_DIS
LIN {X -287.494,Y 38.043,Z 42.917,A -7.538,B 90.000,C 0.000} C_DIS
LIN {X -287.485,Y 38.107,Z 42.968,A -7.551,B 90.000,C 0.000} C_DIS
LIN {X -287.480,Y 38.149,Z 43.019,A -7.559,B 90.000,C 0.000} C_DIS
LIN {X -287.453,Y 38.351,Z 43.061,A -7.599,B 90.000,C 0.000} C_DIS
LIN {X -287.442,Y 38.435,Z 43.164,A -7.616,B 90.000,C 0.000} C_DIS
LIN {X -287.415,Y 38.638,Z 43.206,A -7.656,B 90.000,C 0.000} C_DIS
LIN {X -287.403,Y 38.722,Z 43.308,A -7.673,B 90.000,C 0.000} C_DIS
LIN {X -287.376,Y 38.924,Z 43.350,A -7.714,B 90.000,C 0.000} C_DIS
LIN {X -287.370,Y 38.966,Z 43.402,A -7.722,B 90.000,C 0.000} C_DIS
LIN {X -287.366,Y 38.998,Z 43.453,A -7.728,B 90.000,C 0.000} C_DIS
LIN {X -287.355,Y 39.075,Z 43.474,A -7.744,B 90.000,C 0.000} C_DIS
LIN {X -287.323,Y 39.315,Z 43.639,A -7.791,B 90.000,C 0.000} C_DIS
LIN {X -287.216,Y 40.089,Z 44.410,A -7.946,B 90.000,C 0.000} C_DIS
LIN {X -287.172,Y 40.398,Z 44.847,A -8.007,B 90.000,C 0.000} C_DIS
LIN {X -287.158,Y 40.499,Z 44.958,A -8.028,B 90.000,C 0.000} C_DIS
LIN {X -287.152,Y 40.541,Z 45.080,A -8.036,B 90.000,C 0.000} C_DIS
LIN {X -287.149,Y 40.562,Z 45.170,A -8.040,B 90.000,C 0.000} C_DIS
LIN {X -287.142,Y 40.612,Z 45.208,A -8.050,B 90.000,C 0.000} C_DIS
LIN {X -287.135,Y 40.663,Z 45.272,A -8.060,B 90.000,C 0.000} C_DIS
LIN {X -287.129,Y 40.705,Z 45.578,A -8.069,B 90.000,C 0.000} C_DIS
LIN {X -287.122,Y 40.756,Z 45.642,A -8.079,B 90.000,C 0.000} C_DIS
LIN {X -287.115,Y 40.806,Z 45.727,A -8.089,B 90.000,C 0.000} C_DIS
LIN {X -287.109,Y 40.848,Z 46.135,A -8.097,B 90.000,C 0.000} C_DIS
LIN {X -287.102,Y 40.899,Z 46.220,A -8.107,B 90.000,C 0.000} C_DIS
LIN {X -287.094,Y 40.951,Z 46.473,A -8.118,B 90.000,C 0.000} C_DIS
LIN {X -287.094,Y 40.951,Z 47.846,A -8.118,B 90.000,C 0.000} C_DIS
LIN {X -287.102,Y 40.899,Z 48.099,A -8.107,B 90.000,C 0.000} C_DIS
LIN {X -287.109,Y 40.848,Z 48.184,A -8.097,B 90.000,C 0.000} C_DIS
LIN {X -287.115,Y 40.806,Z 48.592,A -8.089,B 90.000,C 0.000} C_DIS
LIN {X -287.122,Y 40.756,Z 48.677,A -8.079,B 90.000,C 0.000} C_DIS
LIN {X -287.129,Y 40.705,Z 48.740,A -8.069,B 90.000,C 0.000} C_DIS
LIN {X -287.135,Y 40.663,Z 49.047,A -8.060,B 90.000,C 0.000} C_DIS
LIN {X -287.149,Y 40.562,Z 49.174,A -8.040,B 90.000,C 0.000} C_DIS
LIN {X -287.155,Y 40.520,Z 49.480,A -8.032,B 90.000,C 0.000} C_DIS
LIN {X -287.162,Y 40.469,Z 49.544,A -8.022,B 90.000,C 0.000} C_DIS
LIN {X -287.169,Y 40.419,Z 49.586,A -8.012,B 90.000,C 0.000} C_DIS
LIN {X -287.175,Y 40.377,Z 49.791,A -8.003,B 90.000,C 0.000} C_DIS
LIN {X -287.190,Y 40.276,Z 49.875,A -7.983,B 90.000,C 0.000} C_DIS
LIN {X -287.196,Y 40.234,Z 50.080,A -7.975,B 90.000,C 0.000} C_DIS
LIN {X -287.210,Y 40.133,Z 50.165,A -7.955,B 90.000,C 0.000} C_DIS
LIN {X -287.216,Y 40.090,Z 50.369,A -7.946,B 90.000,C 0.000} C_DIS
LIN {X -287.230,Y 39.989,Z 50.449,A -7.926,B 90.000,C 0.000} C_DIS
LIN {X -287.233,Y 39.968,Z 50.540,A -7.922,B 90.000,C 0.000} C_DIS
LIN {X -287.238,Y 39.926,Z 50.661,A -7.913,B 90.000,C 0.000} C_DIS
LIN {X -287.266,Y 39.724,Z 50.884,A -7.873,B 90.000,C 0.000} C_DIS
LIN {X -287.272,Y 39.682,Z 51.005,A -7.865,B 90.000,C 0.000} C_DIS
LIN {X -287.275,Y 39.661,Z 51.096,A -7.861,B 90.000,C 0.000} C_DIS
LIN {X -287.289,Y 39.560,Z 51.172,A -7.840,B 90.000,C 0.000} C_DIS
LIN {X -287.292,Y 39.539,Z 51.262,A -7.836,B 90.000,C 0.000} C_DIS
LIN {X -287.298,Y 39.497,Z 51.384,A -7.828,B 90.000,C 0.000} C_DIS
LIN {X -287.325,Y 39.295,Z 51.606,A -7.787,B 90.000,C 0.000} C_DIS
LIN {X -287.331,Y 39.252,Z 51.728,A -7.779,B 90.000,C 0.000} C_DIS
LIN {X -287.334,Y 39.231,Z 51.819,A -7.775,B 90.000,C 0.000} C_DIS
LIN {X -287.348,Y 39.130,Z 51.899,A -7.755,B 90.000,C 0.000} C_DIS
LIN {X -287.354,Y 39.088,Z 52.103,A -7.746,B 90.000,C 0.000} C_DIS
LIN {X -287.367,Y 38.987,Z 52.183,A -7.726,B 90.000,C 0.000} C_DIS
LIN {X -287.370,Y 38.966,Z 52.274,A -7.722,B 90.000,C 0.000} C_DIS
LIN {X -287.376,Y 38.924,Z 52.395,A -7.714,B 90.000,C 0.000} C_DIS
LIN {X -287.403,Y 38.722,Z 52.618,A -7.673,B 90.000,C 0.000} C_DIS
LIN {X -287.409,Y 38.680,Z 52.740,A -7.665,B 90.000,C 0.000} C_DIS
LIN {X -287.412,Y 38.659,Z 52.830,A -7.661,B 90.000,C 0.000} C_DIS
LIN {X -287.425,Y 38.557,Z 52.906,A -7.640,B 90.000,C 0.000} C_DIS
LIN {X -287.428,Y 38.536,Z 52.997,A -7.636,B 90.000,C 0.000} C_DIS
LIN {X -287.434,Y 38.494,Z 53.118,A -7.628,B 90.000,C 0.000} C_DIS
LIN {X -287.461,Y 38.292,Z 53.341,A -7.588,B 90.000,C 0.000} C_DIS
LIN {X -287.466,Y 38.250,Z 53.462,A -7.579,B 90.000,C 0.000} C_DIS
LIN {X -287.469,Y 38.229,Z 53.553,A -7.575,B 90.000,C 0.000} C_DIS
LIN {X -287.483,Y 38.128,Z 53.629,A -7.555,B 90.000,C 0.000} C_DIS
LIN {X -287.485,Y 38.107,Z 53.719,A -7.551,B 90.000,C 0.000} C_DIS
LIN {X -287.491,Y 38.065,Z 53.841,A -7.542,B 90.000,C 0.000} C_DIS
LIN {X -287.518,Y 37.862,Z 54.063,A -7.502,B 90.000,C 0.000} C_DIS
LIN {X -287.523,Y 37.820,Z 54.185,A -7.494,B 90.000,C 0.000} C_DIS
LIN {X -287.526,Y 37.799,Z 54.276,A -7.489,B 90.000,C 0.000} C_DIS
LIN {X -287.539,Y 37.698,Z 54.351,A -7.469,B 90.000,C 0.000} C_DIS
LIN {X -287.542,Y 37.677,Z 54.442,A -7.465,B 90.000,C 0.000} C_DIS
LIN {X -287.548,Y 37.635,Z 54.563,A -7.457,B 90.000,C 0.000} C_DIS
LIN {X -287.574,Y 37.432,Z 54.786,A -7.416,B 90.000,C 0.000} C_DIS
LIN {X -287.580,Y 37.390,Z 54.907,A -7.408,B 90.000,C 0.000} C_DIS
LIN {X -287.582,Y 37.369,Z 54.998,A -7.404,B 90.000,C 0.000} C_DIS
LIN {X -287.595,Y 37.268,Z 55.074,A -7.383,B 90.000,C 0.000} C_DIS
LIN {X -287.598,Y 37.247,Z 55.165,A -7.379,B 90.000,C 0.000} C_DIS
LIN {X -287.604,Y 37.205,Z 55.286,A -7.371,B 90.000,C 0.000} C_DIS
LIN {X -287.630,Y 37.002,Z 55.509,A -7.331,B 90.000,C 0.000} C_DIS
LIN {X -287.635,Y 36.960,Z 55.630,A -7.322,B 90.000,C 0.000} C_DIS
LIN {X -287.638,Y 36.939,Z 55.721,A -7.318,B 90.000,C 0.000} C_DIS
LIN {X -287.651,Y 36.838,Z 55.796,A -7.298,B 90.000,C 0.000} C_DIS
LIN {X -287.653,Y 36.817,Z 55.887,A -7.294,B 90.000,C 0.000} C_DIS
LIN {X -287.659,Y 36.775,Z 56.009,A -7.285,B 90.000,C 0.000} C_DIS
LIN {X -287.685,Y 36.572,Z 56.231,A -7.245,B 90.000,C 0.000} C_DIS
LIN {X -287.690,Y 36.530,Z 56.353,A -7.237,B 90.000,C 0.000} C_DIS
LIN {X -287.693,Y 36.509,Z 56.444,A -7.232,B 90.000,C 0.000} C_DIS
LIN {X -287.706,Y 36.408,Z 56.519,A -7.212,B 90.000,C 0.000} C_DIS
LIN {X -287.708,Y 36.387,Z 56.610,A -7.208,B 90.000,C 0.000} C_DIS
LIN {X -287.714,Y 36.345,Z 56.731,A -7.200,B 90.000,C 0.000} C_DIS
LIN {X -287.739,Y 36.142,Z 56.954,A -7.159,B 90.000,C 0.000} C_DIS
LIN {X -287.744,Y 36.100,Z 57.075,A -7.151,B 90.000,C 0.000} C_DIS
LIN {X -287.747,Y 36.079,Z 57.166,A -7.147,B 90.000,C 0.000} C_DIS
LIN {X -287.760,Y 35.977,Z 57.242,A -7.126,B 90.000,C 0.000} C_DIS
LIN {X -287.762,Y 35.956,Z 57.333,A -7.122,B 90.000,C 0.000} C_DIS
LIN {X -287.768,Y 35.914,Z 57.454,A -7.114,B 90.000,C 0.000} C_DIS
LIN {X -287.793,Y 35.712,Z 57.677,A -7.074,B 90.000,C 0.000} C_DIS
LIN {X -287.798,Y 35.670,Z 57.798,A -7.065,B 90.000,C 0.000} C_DIS
LIN {X -287.801,Y 35.649,Z 57.889,A -7.061,B 90.000,C 0.000} C_DIS
LIN {X -287.813,Y 35.547,Z 57.969,A -7.041,B 90.000,C 0.000} C_DIS
LIN {X -287.818,Y 35.505,Z 58.173,A -7.032,B 90.000,C 0.000} C_DIS
LIN {X -287.831,Y 35.404,Z 58.253,A -7.012,B 90.000,C 0.000} C_DIS
LIN {X -287.833,Y 35.383,Z 58.344,A -7.008,B 90.000,C 0.000} C_DIS
LIN {X -287.839,Y 35.341,Z 58.466,A -7.000,B 90.000,C 0.000} C_DIS
LIN {X -287.863,Y 35.138,Z 58.688,A -6.959,B 90.000,C 0.000} C_DIS
LIN {X -287.869,Y 35.096,Z 58.810,A -6.951,B 90.000,C 0.000} C_DIS
LIN {X -287.871,Y 35.075,Z 58.901,A -6.947,B 90.000,C 0.000} C_DIS
LIN {X -287.883,Y 34.973,Z 58.976,A -6.927,B 90.000,C 0.000} C_DIS
LIN {X -287.886,Y 34.952,Z 59.067,A -6.922,B 90.000,C 0.000} C_DIS
LIN {X -287.891,Y 34.910,Z 59.188,A -6.914,B 90.000,C 0.000} C_DIS
LIN {X -287.916,Y 34.708,Z 59.411,A -6.874,B 90.000,C 0.000} C_DIS
LIN {X -287.921,Y 34.665,Z 59.532,A -6.865,B 90.000,C 0.000} C_DIS
LIN {X -287.923,Y 34.644,Z 59.623,A -6.861,B 90.000,C 0.000} C_DIS
LIN {X -287.935,Y 34.543,Z 59.699,A -6.841,B 90.000,C 0.000} C_DIS
LIN {X -287.938,Y 34.522,Z 59.790,A -6.837,B 90.000,C 0.000} C_DIS
LIN {X -287.943,Y 34.480,Z 59.911,A -6.828,B 90.000,C 0.000} C_DIS
LIN {X -287.967,Y 34.277,Z 60.134,A -6.788,B 90.000,C 0.000} C_DIS
LIN {X -287.972,Y 34.235,Z 60.255,A -6.780,B 90.000,C 0.000} C_DIS
LIN {X -287.975,Y 34.214,Z 60.346,A -6.775,B 90.000,C 0.000} C_DIS
LIN {X -287.987,Y 34.112,Z 60.421,A -6.755,B 90.000,C 0.000} C_DIS
LIN {X -287.989,Y 34.091,Z 60.512,A -6.751,B 90.000,C 0.000} C_DIS
LIN {X -287.994,Y 34.049,Z 60.634,A -6.743,B 90.000,C 0.000} C_DIS
LIN {X -288.018,Y 33.846,Z 60.856,A -6.702,B 90.000,C 0.000} C_DIS
LIN {X -288.023,Y 33.804,Z 60.978,A -6.694,B 90.000,C 0.000} C_DIS
LIN {X -288.026,Y 33.783,Z 61.068,A -6.690,B 90.000,C 0.000} C_DIS
LIN {X -288.037,Y 33.682,Z 61.144,A -6.670,B 90.000,C 0.000} C_DIS
LIN {X -288.040,Y 33.661,Z 61.235,A -6.665,B 90.000,C 0.000} C_DIS
LIN {X -288.045,Y 33.619,Z 61.356,A -6.657,B 90.000,C 0.000} C_DIS
LIN {X -288.068,Y 33.416,Z 61.579,A -6.617,B 90.000,C 0.000} C_DIS
LIN {X -288.073,Y 33.374,Z 61.700,A -6.608,B 90.000,C 0.000} C_DIS
LIN {X -288.076,Y 33.352,Z 61.791,A -6.604,B 90.000,C 0.000} C_DIS
LIN {X -288.087,Y 33.251,Z 61.867,A -6.584,B 90.000,C 0.000} C_DIS
LIN {X -288.090,Y 33.230,Z 61.957,A -6.580,B 90.000,C 0.000} C_DIS
LIN {X -288.095,Y 33.188,Z 62.079,A -6.571,B 90.000,C 0.000} C_DIS
LIN {X -288.118,Y 32.985,Z 62.302,A -6.531,B 90.000,C 0.000} C_DIS
LIN {X -288.123,Y 32.943,Z 62.423,A -6.523,B 90.000,C 0.000} C_DIS
LIN {X -288.125,Y 32.922,Z 62.514,A -6.518,B 90.000,C 0.000} C_DIS
LIN {X -288.137,Y 32.820,Z 62.589,A -6.498,B 90.000,C 0.000} C_DIS
LIN {X -288.139,Y 32.799,Z 62.680,A -6.494,B 90.000,C 0.000} C_DIS
LIN {X -288.144,Y 32.757,Z 62.801,A -6.486,B 90.000,C 0.000} C_DIS
LIN {X -288.167,Y 32.554,Z 63.024,A -6.445,B 90.000,C 0.000} C_DIS
LIN {X -288.172,Y 32.512,Z 63.146,A -6.437,B 90.000,C 0.000} C_DIS
LIN {X -288.174,Y 32.491,Z 63.236,A -6.433,B 90.000,C 0.000} C_DIS
LIN {X -288.186,Y 32.389,Z 63.312,A -6.413,B 90.000,C 0.000} C_DIS
LIN {X -288.188,Y 32.368,Z 63.403,A -6.408,B 90.000,C 0.000} C_DIS
LIN {X -288.193,Y 32.326,Z 63.524,A -6.400,B 90.000,C 0.000} C_DIS
LIN {X -288.215,Y 32.123,Z 63.747,A -6.360,B 90.000,C 0.000} C_DIS
LIN {X -288.220,Y 32.081,Z 63.868,A -6.351,B 90.000,C 0.000} C_DIS
LIN {X -288.222,Y 32.060,Z 63.959,A -6.347,B 90.000,C 0.000} C_DIS
LIN {X -288.234,Y 31.959,Z 64.035,A -6.327,B 90.000,C 0.000} C_DIS
LIN {X -288.236,Y 31.937,Z 64.125,A -6.323,B 90.000,C 0.000} C_DIS
LIN {X -288.241,Y 31.895,Z 64.247,A -6.314,B 90.000,C 0.000} C_DIS
LIN {X -288.263,Y 31.692,Z 64.469,A -6.274,B 90.000,C 0.000} C_DIS
LIN {X -288.268,Y 31.650,Z 64.591,A -6.266,B 90.000,C 0.000} C_DIS
LIN {X -288.270,Y 31.629,Z 64.682,A -6.261,B 90.000,C 0.000} C_DIS
LIN {X -288.281,Y 31.528,Z 64.757,A -6.241,B 90.000,C 0.000} C_DIS
LIN {X -288.283,Y 31.507,Z 64.848,A -6.237,B 90.000,C 0.000} C_DIS
LIN {X -288.288,Y 31.464,Z 64.969,A -6.229,B 90.000,C 0.000} C_DIS
LIN {X -288.310,Y 31.261,Z 65.192,A -6.188,B 90.000,C 0.000} C_DIS
LIN {X -288.315,Y 31.219,Z 65.314,A -6.180,B 90.000,C 0.000} C_DIS
LIN {X -288.317,Y 31.198,Z 65.404,A -6.176,B 90.000,C 0.000} C_DIS
LIN {X -288.328,Y 31.097,Z 65.485,A -6.156,B 90.000,C 0.000} C_DIS
LIN {X -288.332,Y 31.054,Z 65.689,A -6.147,B 90.000,C 0.000} C_DIS
LIN {X -288.343,Y 30.953,Z 65.769,A -6.127,B 90.000,C 0.000} C_DIS
LIN {X -288.346,Y 30.932,Z 65.860,A -6.123,B 90.000,C 0.000} C_DIS
LIN {X -288.350,Y 30.890,Z 65.981,A -6.114,B 90.000,C 0.000} C_DIS
LIN {X -288.372,Y 30.687,Z 66.204,A -6.074,B 90.000,C 0.000} C_DIS
LIN {X -288.376,Y 30.644,Z 66.325,A -6.066,B 90.000,C 0.000} C_DIS
LIN {X -288.379,Y 30.623,Z 66.416,A -6.062,B 90.000,C 0.000} C_DIS
LIN {X -288.389,Y 30.522,Z 66.492,A -6.041,B 90.000,C 0.000} C_DIS
LIN {X -288.392,Y 30.501,Z 66.582,A -6.037,B 90.000,C 0.000} C_DIS
LIN {X -288.396,Y 30.458,Z 66.704,A -6.029,B 90.000,C 0.000} C_DIS
LIN {X -288.417,Y 30.255,Z 66.926,A -5.988,B 90.000,C 0.000} C_DIS
LIN {X -288.422,Y 30.213,Z 67.048,A -5.980,B 90.000,C 0.000} C_DIS
LIN {X -288.424,Y 30.192,Z 67.139,A -5.976,B 90.000,C 0.000} C_DIS
LIN {X -288.435,Y 30.091,Z 67.214,A -5.956,B 90.000,C 0.000} C_DIS
LIN {X -288.437,Y 30.069,Z 67.305,A -5.952,B 90.000,C 0.000} C_DIS
LIN {X -288.441,Y 30.027,Z 67.426,A -5.943,B 90.000,C 0.000} C_DIS
LIN {X -288.462,Y 29.824,Z 67.649,A -5.903,B 90.000,C 0.000} C_DIS
LIN {X -288.467,Y 29.782,Z 67.770,A -5.894,B 90.000,C 0.000} C_DIS
LIN {X -288.469,Y 29.761,Z 67.861,A -5.890,B 90.000,C 0.000} C_DIS
LIN {X -288.479,Y 29.659,Z 67.937,A -5.870,B 90.000,C 0.000} C_DIS
LIN {X -288.482,Y 29.638,Z 68.028,A -5.866,B 90.000,C 0.000} C_DIS
LIN {X -288.486,Y 29.596,Z 68.149,A -5.858,B 90.000,C 0.000} C_DIS
LIN {X -288.507,Y 29.393,Z 68.372,A -5.817,B 90.000,C 0.000} C_DIS
LIN {X -288.511,Y 29.351,Z 68.493,A -5.809,B 90.000,C 0.000} C_DIS
LIN {X -288.513,Y 29.329,Z 68.584,A -5.805,B 90.000,C 0.000} C_DIS
LIN {X -288.523,Y 29.228,Z 68.659,A -5.784,B 90.000,C 0.000} C_DIS
LIN {X -288.526,Y 29.207,Z 68.750,A -5.780,B 90.000,C 0.000} C_DIS
LIN {X -288.530,Y 29.165,Z 68.872,A -5.772,B 90.000,C 0.000} C_DIS
LIN {X -288.550,Y 28.961,Z 69.094,A -5.732,B 90.000,C 0.000} C_DIS
LIN {X -288.554,Y 28.919,Z 69.216,A -5.723,B 90.000,C 0.000} C_DIS
LIN {X -288.557,Y 28.898,Z 69.307,A -5.719,B 90.000,C 0.000} C_DIS
LIN {X -288.567,Y 28.796,Z 69.382,A -5.699,B 90.000,C 0.000} C_DIS
LIN {X -288.569,Y 28.775,Z 69.473,A -5.695,B 90.000,C 0.000} C_DIS
LIN {X -288.573,Y 28.733,Z 69.594,A -5.686,B 90.000,C 0.000} C_DIS
LIN {X -288.593,Y 28.530,Z 69.817,A -5.646,B 90.000,C 0.000} C_DIS
LIN {X -288.597,Y 28.488,Z 69.938,A -5.637,B 90.000,C 0.000} C_DIS
LIN {X -288.599,Y 28.467,Z 70.029,A -5.633,B 90.000,C 0.000} C_DIS
LIN {X -288.609,Y 28.365,Z 70.105,A -5.613,B 90.000,C 0.000} C_DIS
LIN {X -288.612,Y 28.344,Z 70.196,A -5.609,B 90.000,C 0.000} C_DIS
LIN {X -288.616,Y 28.302,Z 70.317,A -5.601,B 90.000,C 0.000} C_DIS
LIN {X -288.636,Y 28.098,Z 70.540,A -5.560,B 90.000,C 0.000} C_DIS
LIN {X -288.640,Y 28.056,Z 70.661,A -5.552,B 90.000,C 0.000} C_DIS
LIN {X -288.642,Y 28.035,Z 70.752,A -5.548,B 90.000,C 0.000} C_DIS
LIN {X -288.652,Y 27.933,Z 70.832,A -5.527,B 90.000,C 0.000} C_DIS
LIN {X -288.656,Y 27.891,Z 71.036,A -5.519,B 90.000,C 0.000} C_DIS
LIN {X -288.665,Y 27.790,Z 71.116,A -5.499,B 90.000,C 0.000} C_DIS
LIN {X -288.667,Y 27.768,Z 71.207,A -5.495,B 90.000,C 0.000} C_DIS
LIN {X -288.672,Y 27.726,Z 71.329,A -5.486,B 90.000,C 0.000} C_DIS
LIN {X -288.691,Y 27.523,Z 71.551,A -5.446,B 90.000,C 0.000} C_DIS
LIN {X -288.695,Y 27.481,Z 71.673,A -5.438,B 90.000,C 0.000} C_DIS
LIN {X -288.697,Y 27.460,Z 71.764,A -5.433,B 90.000,C 0.000} C_DIS
LIN {X -288.707,Y 27.358,Z 71.839,A -5.413,B 90.000,C 0.000} C_DIS
LIN {X -288.709,Y 27.337,Z 71.930,A -5.409,B 90.000,C 0.000} C_DIS
LIN {X -288.713,Y 27.295,Z 72.051,A -5.401,B 90.000,C 0.000} C_DIS
LIN {X -288.732,Y 27.091,Z 72.274,A -5.360,B 90.000,C 0.000} C_DIS
LIN {X -288.736,Y 27.049,Z 72.395,A -5.352,B 90.000,C 0.000} C_DIS
LIN {X -288.738,Y 27.028,Z 72.486,A -5.348,B 90.000,C 0.000} C_DIS
LIN {X -288.747,Y 26.926,Z 72.562,A -5.328,B 90.000,C 0.000} C_DIS
LIN {X -288.749,Y 26.905,Z 72.653,A -5.323,B 90.000,C 0.000} C_DIS
LIN {X -288.753,Y 26.863,Z 72.774,A -5.315,B 90.000,C 0.000} C_DIS
LIN {X -288.772,Y 26.660,Z 72.997,A -5.275,B 90.000,C 0.000} C_DIS
LIN {X -288.776,Y 26.617,Z 73.118,A -5.266,B 90.000,C 0.000} C_DIS
LIN {X -288.778,Y 26.596,Z 73.209,A -5.262,B 90.000,C 0.000} C_DIS
LIN {X -288.787,Y 26.495,Z 73.284,A -5.242,B 90.000,C 0.000} C_DIS
LIN {X -288.789,Y 26.473,Z 73.375,A -5.238,B 90.000,C 0.000} C_DIS
LIN {X -288.793,Y 26.431,Z 73.497,A -5.229,B 90.000,C 0.000} C_DIS
LIN {X -288.812,Y 26.228,Z 73.719,A -5.189,B 90.000,C 0.000} C_DIS
LIN {X -288.815,Y 26.186,Z 73.841,A -5.181,B 90.000,C 0.000} C_DIS
LIN {X -288.817,Y 26.164,Z 73.931,A -5.176,B 90.000,C 0.000} C_DIS
LIN {X -288.826,Y 26.063,Z 74.007,A -5.156,B 90.000,C 0.000} C_DIS
LIN {X -288.828,Y 26.042,Z 74.098,A -5.152,B 90.000,C 0.000} C_DIS
LIN {X -288.832,Y 25.999,Z 74.219,A -5.144,B 90.000,C 0.000} C_DIS
LIN {X -288.850,Y 25.796,Z 74.442,A -5.103,B 90.000,C 0.000} C_DIS
LIN {X -288.854,Y 25.754,Z 74.563,A -5.095,B 90.000,C 0.000} C_DIS
LIN {X -288.856,Y 25.733,Z 74.654,A -5.091,B 90.000,C 0.000} C_DIS
LIN {X -288.865,Y 25.631,Z 74.730,A -5.071,B 90.000,C 0.000} C_DIS
LIN {X -288.867,Y 25.610,Z 74.820,A -5.066,B 90.000,C 0.000} C_DIS
LIN {X -288.871,Y 25.567,Z 74.942,A -5.058,B 90.000,C 0.000} C_DIS
LIN {X -288.889,Y 25.364,Z 75.165,A -5.018,B 90.000,C 0.000} C_DIS
LIN {X -288.892,Y 25.322,Z 75.286,A -5.009,B 90.000,C 0.000} C_DIS
LIN {X -288.894,Y 25.301,Z 75.377,A -5.005,B 90.000,C 0.000} C_DIS
LIN {X -288.903,Y 25.199,Z 75.452,A -4.985,B 90.000,C 0.000} C_DIS
LIN {X -288.905,Y 25.178,Z 75.543,A -4.981,B 90.000,C 0.000} C_DIS
LIN {X -288.909,Y 25.136,Z 75.665,A -4.972,B 90.000,C 0.000} C_DIS
LIN {X -288.926,Y 24.932,Z 75.887,A -4.932,B 90.000,C 0.000} C_DIS
LIN {X -288.930,Y 24.890,Z 76.009,A -4.924,B 90.000,C 0.000} C_DIS
LIN {X -288.932,Y 24.869,Z 76.099,A -4.919,B 90.000,C 0.000} C_DIS
LIN {X -288.940,Y 24.767,Z 76.175,A -4.899,B 90.000,C 0.000} C_DIS
LIN {X -288.942,Y 24.746,Z 76.266,A -4.895,B 90.000,C 0.000} C_DIS
LIN {X -288.946,Y 24.704,Z 76.387,A -4.887,B 90.000,C 0.000} C_DIS
LIN {X -288.963,Y 24.500,Z 76.610,A -4.846,B 90.000,C 0.000} C_DIS
LIN {X -288.967,Y 24.458,Z 76.731,A -4.838,B 90.000,C 0.000} C_DIS
LIN {X -288.969,Y 24.437,Z 76.822,A -4.834,B 90.000,C 0.000} C_DIS
LIN {X -288.977,Y 24.335,Z 76.902,A -4.814,B 90.000,C 0.000} C_DIS
LIN {X -288.981,Y 24.293,Z 77.106,A -4.805,B 90.000,C 0.000} C_DIS
LIN {X -288.989,Y 24.191,Z 77.187,A -4.785,B 90.000,C 0.000} C_DIS
LIN {X -288.991,Y 24.170,Z 77.277,A -4.781,B 90.000,C 0.000} C_DIS
LIN {X -288.995,Y 24.127,Z 77.399,A -4.772,B 90.000,C 0.000} C_DIS
LIN {X -289.011,Y 23.924,Z 77.622,A -4.732,B 90.000,C 0.000} C_DIS
LIN {X -289.015,Y 23.882,Z 77.743,A -4.724,B 90.000,C 0.000} C_DIS
LIN {X -289.017,Y 23.861,Z 77.834,A -4.720,B 90.000,C 0.000} C_DIS
LIN {X -289.025,Y 23.759,Z 77.909,A -4.699,B 90.000,C 0.000} C_DIS
LIN {X -289.027,Y 23.738,Z 78.000,A -4.695,B 90.000,C 0.000} C_DIS
LIN {X -289.030,Y 23.695,Z 78.121,A -4.687,B 90.000,C 0.000} C_DIS
LIN {X -289.047,Y 23.492,Z 78.344,A -4.646,B 90.000,C 0.000} C_DIS
LIN {X -289.050,Y 23.450,Z 78.466,A -4.638,B 90.000,C 0.000} C_DIS
LIN {X -289.052,Y 23.428,Z 78.556,A -4.634,B 90.000,C 0.000} C_DIS
LIN {X -289.060,Y 23.327,Z 78.632,A -4.614,B 90.000,C 0.000} C_DIS
LIN {X -289.062,Y 23.306,Z 78.723,A -4.609,B 90.000,C 0.000} C_DIS
LIN {X -289.065,Y 23.263,Z 78.844,A -4.601,B 90.000,C 0.000} C_DIS
LIN {X -289.082,Y 23.060,Z 79.067,A -4.561,B 90.000,C 0.000} C_DIS
LIN {X -289.085,Y 23.017,Z 79.188,A -4.552,B 90.000,C 0.000} C_DIS
LIN {X -289.087,Y 22.996,Z 79.279,A -4.548,B 90.000,C 0.000} C_DIS
LIN {X -289.095,Y 22.894,Z 79.355,A -4.528,B 90.000,C 0.000} C_DIS
LIN {X -289.097,Y 22.873,Z 79.445,A -4.524,B 90.000,C 0.000} C_DIS
LIN {X -289.100,Y 22.831,Z 79.567,A -4.515,B 90.000,C 0.000} C_DIS
LIN {X -289.116,Y 22.627,Z 79.789,A -4.475,B 90.000,C 0.000} C_DIS
LIN {X -289.119,Y 22.585,Z 79.911,A -4.467,B 90.000,C 0.000} C_DIS
LIN {X -289.121,Y 22.564,Z 80.002,A -4.463,B 90.000,C 0.000} C_DIS
LIN {X -289.129,Y 22.462,Z 80.077,A -4.442,B 90.000,C 0.000} C_DIS
LIN {X -289.130,Y 22.441,Z 80.168,A -4.438,B 90.000,C 0.000} C_DIS
LIN {X -289.134,Y 22.399,Z 80.289,A -4.430,B 90.000,C 0.000} C_DIS
LIN {X -289.149,Y 22.195,Z 80.512,A -4.389,B 90.000,C 0.000} C_DIS
LIN {X -289.153,Y 22.153,Z 80.633,A -4.381,B 90.000,C 0.000} C_DIS
LIN {X -289.154,Y 22.132,Z 80.724,A -4.377,B 90.000,C 0.000} C_DIS
LIN {X -289.162,Y 22.030,Z 80.800,A -4.357,B 90.000,C 0.000} C_DIS
LIN {X -289.164,Y 22.009,Z 80.891,A -4.352,B 90.000,C 0.000} C_DIS
LIN {X -289.167,Y 21.966,Z 81.012,A -4.344,B 90.000,C 0.000} C_DIS
LIN {X -289.182,Y 21.763,Z 81.235,A -4.304,B 90.000,C 0.000} C_DIS
LIN {X -289.185,Y 21.721,Z 81.356,A -4.295,B 90.000,C 0.000} C_DIS
LIN {X -289.187,Y 21.699,Z 81.447,A -4.291,B 90.000,C 0.000} C_DIS
LIN {X -289.195,Y 21.598,Z 81.522,A -4.271,B 90.000,C 0.000} C_DIS
LIN {X -289.196,Y 21.576,Z 81.613,A -4.267,B 90.000,C 0.000} C_DIS
LIN {X -289.199,Y 21.534,Z 81.735,A -4.258,B 90.000,C 0.000} C_DIS
LIN {X -289.214,Y 21.330,Z 81.957,A -4.218,B 90.000,C 0.000} C_DIS
LIN {X -289.218,Y 21.288,Z 82.079,A -4.210,B 90.000,C 0.000} C_DIS
LIN {X -289.219,Y 21.267,Z 82.170,A -4.206,B 90.000,C 0.000} C_DIS
LIN {X -289.227,Y 21.165,Z 82.245,A -4.185,B 90.000,C 0.000} C_DIS
LIN {X -289.228,Y 21.144,Z 82.336,A -4.181,B 90.000,C 0.000} C_DIS
LIN {X -289.231,Y 21.102,Z 82.457,A -4.173,B 90.000,C 0.000} C_DIS
LIN {X -289.246,Y 20.898,Z 82.680,A -4.132,B 90.000,C 0.000} C_DIS
LIN {X -289.249,Y 20.856,Z 82.801,A -4.124,B 90.000,C 0.000} C_DIS
LIN {X -289.251,Y 20.835,Z 82.892,A -4.120,B 90.000,C 0.000} C_DIS
LIN {X -289.258,Y 20.733,Z 82.968,A -4.100,B 90.000,C 0.000} C_DIS
LIN {X -289.259,Y 20.712,Z 83.059,A -4.096,B 90.000,C 0.000} C_DIS
LIN {X -289.262,Y 20.669,Z 83.180,A -4.087,B 90.000,C 0.000} C_DIS
LIN {X -289.277,Y 20.466,Z 83.403,A -4.047,B 90.000,C 0.000} C_DIS
LIN {X -289.280,Y 20.423,Z 83.524,A -4.038,B 90.000,C 0.000} C_DIS
LIN {X -289.281,Y 20.402,Z 83.615,A -4.034,B 90.000,C 0.000} C_DIS
LIN {X -289.289,Y 20.300,Z 83.695,A -4.014,B 90.000,C 0.000} C_DIS
LIN {X -289.292,Y 20.258,Z 83.899,A -4.006,B 90.000,C 0.000} C_DIS
LIN {X -289.299,Y 20.156,Z 83.979,A -3.985,B 90.000,C 0.000} C_DIS
LIN {X -289.300,Y 20.135,Z 84.070,A -3.981,B 90.000,C 0.000} C_DIS
LIN {X -289.303,Y 20.093,Z 84.192,A -3.973,B 90.000,C 0.000} C_DIS
LIN {X -289.317,Y 19.889,Z 84.414,A -3.933,B 90.000,C 0.000} C_DIS
LIN {X -289.320,Y 19.846,Z 84.536,A -3.924,B 90.000,C 0.000} C_DIS
LIN {X -289.322,Y 19.825,Z 84.627,A -3.920,B 90.000,C 0.000} C_DIS
LIN {X -289.329,Y 19.723,Z 84.702,A -3.900,B 90.000,C 0.000} C_DIS
LIN {X -289.330,Y 19.702,Z 84.793,A -3.896,B 90.000,C 0.000} C_DIS
LIN {X -289.333,Y 19.660,Z 84.914,A -3.887,B 90.000,C 0.000} C_DIS
LIN {X -289.347,Y 19.456,Z 85.137,A -3.847,B 90.000,C 0.000} C_DIS
LIN {X -289.349,Y 19.414,Z 85.258,A -3.839,B 90.000,C 0.000} C_DIS
LIN {X -289.351,Y 19.393,Z 85.349,A -3.834,B 90.000,C 0.000} C_DIS
LIN {X -289.358,Y 19.291,Z 85.425,A -3.814,B 90.000,C 0.000} C_DIS
LIN {X -289.359,Y 19.270,Z 85.516,A -3.810,B 90.000,C 0.000} C_DIS
LIN {X -289.362,Y 19.227,Z 85.637,A -3.802,B 90.000,C 0.000} C_DIS
LIN {X -289.375,Y 19.024,Z 85.860,A -3.761,B 90.000,C 0.000} C_DIS
LIN {X -289.378,Y 18.981,Z 85.981,A -3.753,B 90.000,C 0.000} C_DIS
LIN {X -289.380,Y 18.960,Z 86.072,A -3.749,B 90.000,C 0.000} C_DIS
LIN {X -289.386,Y 18.858,Z 86.147,A -3.728,B 90.000,C 0.000} C_DIS
LIN {X -289.388,Y 18.837,Z 86.238,A -3.724,B 90.000,C 0.000} C_DIS
LIN {X -289.390,Y 18.795,Z 86.360,A -3.716,B 90.000,C 0.000} C_DIS
LIN {X -289.403,Y 18.591,Z 86.582,A -3.676,B 90.000,C 0.000} C_DIS
LIN {X -289.406,Y 18.549,Z 86.704,A -3.667,B 90.000,C 0.000} C_DIS
LIN {X -289.408,Y 18.527,Z 86.794,A -3.663,B 90.000,C 0.000} C_DIS
LIN {X -289.414,Y 18.426,Z 86.870,A -3.643,B 90.000,C 0.000} C_DIS
LIN {X -289.415,Y 18.404,Z 86.961,A -3.639,B 90.000,C 0.000} C_DIS
LIN {X -289.418,Y 18.362,Z 87.082,A -3.630,B 90.000,C 0.000} C_DIS
LIN {X -289.431,Y 18.158,Z 87.305,A -3.590,B 90.000,C 0.000} C_DIS
LIN {X -289.434,Y 18.116,Z 87.426,A -3.582,B 90.000,C 0.000} C_DIS
LIN {X -289.435,Y 18.095,Z 87.517,A -3.577,B 90.000,C 0.000} C_DIS
LIN {X -289.441,Y 17.993,Z 87.593,A -3.557,B 90.000,C 0.000} C_DIS
LIN {X -289.443,Y 17.972,Z 87.683,A -3.553,B 90.000,C 0.000} C_DIS
LIN {X -289.445,Y 17.929,Z 87.805,A -3.545,B 90.000,C 0.000} C_DIS
LIN {X -289.458,Y 17.725,Z 88.028,A -3.504,B 90.000,C 0.000} C_DIS
LIN {X -289.460,Y 17.683,Z 88.149,A -3.496,B 90.000,C 0.000} C_DIS
LIN {X -289.462,Y 17.662,Z 88.240,A -3.492,B 90.000,C 0.000} C_DIS
LIN {X -289.468,Y 17.560,Z 88.315,A -3.471,B 90.000,C 0.000} C_DIS
LIN {X -289.469,Y 17.539,Z 88.406,A -3.467,B 90.000,C 0.000} C_DIS
LIN {X -289.472,Y 17.496,Z 88.528,A -3.459,B 90.000,C 0.000} C_DIS
LIN {X -289.484,Y 17.293,Z 88.750,A -3.419,B 90.000,C 0.000} C_DIS
LIN {X -289.486,Y 17.250,Z 88.872,A -3.410,B 90.000,C 0.000} C_DIS
LIN {X -289.488,Y 17.229,Z 88.962,A -3.406,B 90.000,C 0.000} C_DIS
LIN {X -289.494,Y 17.127,Z 89.038,A -3.386,B 90.000,C 0.000} C_DIS
LIN {X -289.495,Y 17.106,Z 89.129,A -3.382,B 90.000,C 0.000} C_DIS
LIN {X -289.498,Y 17.064,Z 89.250,A -3.373,B 90.000,C 0.000} C_DIS
LIN {X -289.509,Y 16.860,Z 89.473,A -3.333,B 90.000,C 0.000} C_DIS
LIN {X -289.512,Y 16.817,Z 89.594,A -3.325,B 90.000,C 0.000} C_DIS
LIN {X -289.513,Y 16.796,Z 89.685,A -3.320,B 90.000,C 0.000} C_DIS
LIN {X -289.519,Y 16.694,Z 89.765,A -3.300,B 90.000,C 0.000} C_DIS
LIN {X -289.522,Y 16.652,Z 89.969,A -3.292,B 90.000,C 0.000} C_DIS
LIN {X -289.527,Y 16.550,Z 90.050,A -3.272,B 90.000,C 0.000} C_DIS
LIN {X -289.529,Y 16.529,Z 90.140,A -3.267,B 90.000,C 0.000} C_DIS
LIN {X -289.531,Y 16.487,Z 90.262,A -3.259,B 90.000,C 0.000} C_DIS
LIN {X -289.543,Y 16.283,Z 90.485,A -3.219,B 90.000,C 0.000} C_DIS
LIN {X -289.545,Y 16.240,Z 90.606,A -3.210,B 90.000,C 0.000} C_DIS
LIN {X -289.546,Y 16.219,Z 90.697,A -3.206,B 90.000,C 0.000} C_DIS
LIN {X -289.552,Y 16.117,Z 90.772,A -3.186,B 90.000,C 0.000} C_DIS
LIN {X -289.553,Y 16.096,Z 90.863,A -3.182,B 90.000,C 0.000} C_DIS
LIN {X -289.555,Y 16.054,Z 90.984,A -3.173,B 90.000,C 0.000} C_DIS
LIN {X -289.567,Y 15.850,Z 91.207,A -3.133,B 90.000,C 0.000} C_DIS
LIN {X -289.569,Y 15.807,Z 91.329,A -3.125,B 90.000,C 0.000} C_DIS
LIN {X -289.570,Y 15.786,Z 91.419,A -3.120,B 90.000,C 0.000} C_DIS
LIN {X -289.576,Y 15.684,Z 91.495,A -3.100,B 90.000,C 0.000} C_DIS
LIN {X -289.577,Y 15.663,Z 91.586,A -3.096,B 90.000,C 0.000} C_DIS
LIN {X -289.579,Y 15.621,Z 91.707,A -3.088,B 90.000,C 0.000} C_DIS
LIN {X -289.590,Y 15.417,Z 91.930,A -3.047,B 90.000,C 0.000} C_DIS
LIN {X -289.592,Y 15.374,Z 92.051,A -3.039,B 90.000,C 0.000} C_DIS
LIN {X -289.593,Y 15.353,Z 92.142,A -3.035,B 90.000,C 0.000} C_DIS
LIN {X -289.599,Y 15.251,Z 92.218,A -3.015,B 90.000,C 0.000} C_DIS
LIN {X -289.600,Y 15.230,Z 92.308,A -3.010,B 90.000,C 0.000} C_DIS
LIN {X -289.602,Y 15.188,Z 92.430,A -3.002,B 90.000,C 0.000} C_DIS
LIN {X -289.613,Y 14.984,Z 92.652,A -2.962,B 90.000,C 0.000} C_DIS
LIN {X -289.615,Y 14.941,Z 92.774,A -2.953,B 90.000,C 0.000} C_DIS
LIN {X -289.616,Y 14.920,Z 92.865,A -2.949,B 90.000,C 0.000} C_DIS
LIN {X -289.621,Y 14.818,Z 92.940,A -2.929,B 90.000,C 0.000} C_DIS
LIN {X -289.622,Y 14.797,Z 93.031,A -2.925,B 90.000,C 0.000} C_DIS
LIN {X -289.624,Y 14.755,Z 93.152,A -2.916,B 90.000,C 0.000} C_DIS
LIN {X -289.635,Y 14.551,Z 93.375,A -2.876,B 90.000,C 0.000} C_DIS
LIN {X -289.637,Y 14.508,Z 93.497,A -2.868,B 90.000,C 0.000} C_DIS
LIN {X -289.638,Y 14.487,Z 93.587,A -2.863,B 90.000,C 0.000} C_DIS
LIN {X -289.643,Y 14.385,Z 93.663,A -2.843,B 90.000,C 0.000} C_DIS
LIN {X -289.644,Y 14.364,Z 93.754,A -2.839,B 90.000,C 0.000} C_DIS
LIN {X -289.646,Y 14.322,Z 93.875,A -2.831,B 90.000,C 0.000} C_DIS
LIN {X -289.656,Y 14.118,Z 94.098,A -2.790,B 90.000,C 0.000} C_DIS
LIN {X -289.658,Y 14.075,Z 94.219,A -2.782,B 90.000,C 0.000} C_DIS
LIN {X -289.659,Y 14.054,Z 94.310,A -2.778,B 90.000,C 0.000} C_DIS
LIN {X -289.664,Y 13.952,Z 94.385,A -2.758,B 90.000,C 0.000} C_DIS
LIN {X -289.665,Y 13.931,Z 94.476,A -2.753,B 90.000,C 0.000} C_DIS
LIN {X -289.667,Y 13.889,Z 94.598,A -2.745,B 90.000,C 0.000} C_DIS
LIN {X -289.677,Y 13.685,Z 94.820,A -2.705,B 90.000,C 0.000} C_DIS
LIN {X -289.679,Y 13.642,Z 94.942,A -2.696,B 90.000,C 0.000} C_DIS
LIN {X -289.680,Y 13.621,Z 95.033,A -2.692,B 90.000,C 0.000} C_DIS
LIN {X -289.685,Y 13.519,Z 95.108,A -2.672,B 90.000,C 0.000} C_DIS
LIN {X -289.686,Y 13.498,Z 95.199,A -2.668,B 90.000,C 0.000} C_DIS
LIN {X -289.688,Y 13.455,Z 95.320,A -2.659,B 90.000,C 0.000} C_DIS
LIN {X -289.697,Y 13.252,Z 95.543,A -2.619,B 90.000,C 0.000} C_DIS
LIN {X -289.699,Y 13.209,Z 95.664,A -2.611,B 90.000,C 0.000} C_DIS
LIN {X -289.700,Y 13.188,Z 95.755,A -2.606,B 90.000,C 0.000} C_DIS
LIN {X -289.705,Y 13.086,Z 95.831,A -2.586,B 90.000,C 0.000} C_DIS
LIN {X -289.706,Y 13.065,Z 95.922,A -2.582,B 90.000,C 0.000} C_DIS
LIN {X -289.707,Y 13.022,Z 96.043,A -2.574,B 90.000,C 0.000} C_DIS
LIN {X -289.717,Y 12.818,Z 96.266,A -2.533,B 90.000,C 0.000} C_DIS
LIN {X -289.718,Y 12.776,Z 96.387,A -2.525,B 90.000,C 0.000} C_DIS
LIN {X -289.719,Y 12.755,Z 96.478,A -2.521,B 90.000,C 0.000} C_DIS
LIN {X -289.724,Y 12.653,Z 96.558,A -2.501,B 90.000,C 0.000} C_DIS
LIN {X -289.726,Y 12.610,Z 96.762,A -2.492,B 90.000,C 0.000} C_DIS
LIN {X -289.730,Y 12.508,Z 96.842,A -2.472,B 90.000,C 0.000} C_DIS
LIN {X -289.731,Y 12.487,Z 96.933,A -2.468,B 90.000,C 0.000} C_DIS
LIN {X -289.733,Y 12.445,Z 97.055,A -2.459,B 90.000,C 0.000} C_DIS
LIN {X -289.742,Y 12.241,Z 97.277,A -2.419,B 90.000,C 0.000} C_DIS
LIN {X -289.743,Y 12.198,Z 97.399,A -2.411,B 90.000,C 0.000} C_DIS
LIN {X -289.744,Y 12.177,Z 97.490,A -2.407,B 90.000,C 0.000} C_DIS
LIN {X -289.748,Y 12.075,Z 97.565,A -2.386,B 90.000,C 0.000} C_DIS
LIN {X -289.749,Y 12.054,Z 97.656,A -2.382,B 90.000,C 0.000} C_DIS
LIN {X -289.751,Y 12.012,Z 97.777,A -2.374,B 90.000,C 0.000} C_DIS
LIN {X -289.760,Y 11.808,Z 98.000,A -2.333,B 90.000,C 0.000} C_DIS
LIN {X -289.761,Y 11.765,Z 98.121,A -2.325,B 90.000,C 0.000} C_DIS
LIN {X -289.762,Y 11.744,Z 98.212,A -2.321,B 90.000,C 0.000} C_DIS
LIN {X -289.766,Y 11.642,Z 98.288,A -2.301,B 90.000,C 0.000} C_DIS
LIN {X -289.767,Y 11.621,Z 98.379,A -2.297,B 90.000,C 0.000} C_DIS
LIN {X -289.769,Y 11.578,Z 98.500,A -2.288,B 90.000,C 0.000} C_DIS
LIN {X -289.777,Y 11.374,Z 98.723,A -2.248,B 90.000,C 0.000} C_DIS
LIN {X -289.779,Y 11.332,Z 98.844,A -2.239,B 90.000,C 0.000} C_DIS
LIN {X -289.779,Y 11.311,Z 98.935,A -2.235,B 90.000,C 0.000} C_DIS
LIN {X -289.783,Y 11.209,Z 99.010,A -2.215,B 90.000,C 0.000} C_DIS
LIN {X -289.784,Y 11.188,Z 99.101,A -2.211,B 90.000,C 0.000} C_DIS
LIN {X -289.786,Y 11.145,Z 99.223,A -2.203,B 90.000,C 0.000} C_DIS
LIN {X -289.794,Y 10.941,Z 99.445,A -2.162,B 90.000,C 0.000} C_DIS
LIN {X -289.795,Y 10.899,Z 99.567,A -2.154,B 90.000,C 0.000} C_DIS
LIN {X -289.796,Y 10.877,Z 99.657,A -2.150,B 90.000,C 0.000} C_DIS
LIN {X -289.800,Y 10.775,Z 99.733,A -2.129,B 90.000,C 0.000} C_DIS
LIN {X -289.801,Y 10.754,Z 99.824,A -2.125,B 90.000,C 0.000} C_DIS
LIN {X -289.802,Y 10.712,Z 99.945,A -2.117,B 90.000,C 0.000} C_DIS
LIN {X -289.810,Y 10.508,Z 100.168,A -2.077,B 90.000,C 0.000} C_DIS
LIN {X -289.811,Y 10.465,Z 100.289,A -2.068,B 90.000,C 0.000} C_DIS
LIN {X -289.812,Y 10.444,Z 100.380,A -2.064,B 90.000,C 0.000} C_DIS
LIN {X -289.816,Y 10.342,Z 100.456,A -2.044,B 90.000,C 0.000} C_DIS
LIN {X -289.816,Y 10.321,Z 100.546,A -2.040,B 90.000,C 0.000} C_DIS
LIN {X -289.818,Y 10.279,Z 100.668,A -2.031,B 90.000,C 0.000} C_DIS
LIN {X -289.825,Y 10.075,Z 100.891,A -1.991,B 90.000,C 0.000} C_DIS
LIN {X -289.826,Y 10.032,Z 101.012,A -1.982,B 90.000,C 0.000} C_DIS
LIN {X -289.827,Y 10.011,Z 101.103,A -1.978,B 90.000,C 0.000} C_DIS
LIN {X -289.831,Y 9.909,Z 101.178,A -1.958,B 90.000,C 0.000} C_DIS
LIN {X -289.831,Y 9.888,Z 101.269,A -1.954,B 90.000,C 0.000} C_DIS
LIN {X -289.833,Y 9.845,Z 101.391,A -1.946,B 90.000,C 0.000} C_DIS
LIN {X -289.840,Y 9.641,Z 101.613,A -1.905,B 90.000,C 0.000} C_DIS
LIN {X -289.841,Y 9.599,Z 101.735,A -1.897,B 90.000,C 0.000} C_DIS
LIN {X -289.842,Y 9.578,Z 101.825,A -1.893,B 90.000,C 0.000} C_DIS
LIN {X -289.845,Y 9.476,Z 101.901,A -1.872,B 90.000,C 0.000} C_DIS
LIN {X -289.846,Y 9.454,Z 101.992,A -1.868,B 90.000,C 0.000} C_DIS
LIN {X -289.847,Y 9.412,Z 102.113,A -1.860,B 90.000,C 0.000} C_DIS
LIN {X -289.854,Y 9.208,Z 102.336,A -1.820,B 90.000,C 0.000} C_DIS
LIN {X -289.855,Y 9.165,Z 102.457,A -1.811,B 90.000,C 0.000} C_DIS
LIN {X -289.856,Y 9.144,Z 102.548,A -1.807,B 90.000,C 0.000} C_DIS
LIN {X -289.859,Y 9.042,Z 102.628,A -1.787,B 90.000,C 0.000} C_DIS
LIN {X -289.860,Y 9.000,Z 102.832,A -1.778,B 90.000,C 0.000} C_DIS
LIN {X -289.863,Y 8.898,Z 102.913,A -1.758,B 90.000,C 0.000} C_DIS
LIN {X -289.864,Y 8.876,Z 103.003,A -1.754,B 90.000,C 0.000} C_DIS
LIN {X -289.865,Y 8.834,Z 103.125,A -1.746,B 90.000,C 0.000} C_DIS
LIN {X -289.872,Y 8.630,Z 103.348,A -1.705,B 90.000,C 0.000} C_DIS
LIN {X -289.873,Y 8.588,Z 103.469,A -1.697,B 90.000,C 0.000} C_DIS
LIN {X -289.873,Y 8.566,Z 103.560,A -1.693,B 90.000,C 0.000} C_DIS
LIN {X -289.876,Y 8.464,Z 103.635,A -1.673,B 90.000,C 0.000} C_DIS
LIN {X -289.877,Y 8.443,Z 103.726,A -1.668,B 90.000,C 0.000} C_DIS
LIN {X -289.878,Y 8.401,Z 103.848,A -1.660,B 90.000,C 0.000} C_DIS
LIN {X -289.884,Y 8.197,Z 104.070,A -1.620,B 90.000,C 0.000} C_DIS
LIN {X -289.885,Y 8.154,Z 104.192,A -1.611,B 90.000,C 0.000} C_DIS
LIN {X -289.886,Y 8.133,Z 104.282,A -1.607,B 90.000,C 0.000} C_DIS
LIN {X -289.889,Y 8.031,Z 104.354,A -1.587,B 90.000,C 0.000} C_DIS
LIN {X -289.890,Y 7.976,Z 104.549,A -1.576,B 90.000,C 0.000} C_DIS
LIN {X -289.892,Y 7.898,Z 104.656,A -1.561,B 90.000,C 0.000} C_DIS
RET=EKI_SetBool("oxy","torchState",FALSE)
RET = EKI_Send("oxy","torchState")
PTP {X -287.893,Y 7.844,Z 104.656,A -1.561,B 90.000,C 0.000}
PTP {X -269.900,Y 7.353,Z 104.656,A -1.561,B 90.000,C 0.000}
PTP {X -269.885,Y -7.886,Z 104.668,A 1.674,B 90.000,C 0.000}
PTP {X -287.877,Y -8.411,Z 104.668,A 1.674,B 90.000,C 0.000}
WAIT SEC 2
RET=EKI_SetBool("oxy","torchState",TRUE)
RET = EKI_Send("oxy","torchState")
LIN {X -289.876,Y -8.470,Z 104.668,A 1.674,B 90.000,C 0.000} C_DIS
LIN {X -289.876,Y -8.479,Z 104.716,A 1.675,B 90.000,C 0.000} C_DIS
LIN {X -289.874,Y -8.550,Z 104.723,A 1.690,B 90.000,C 0.000} C_DIS
LIN {X -289.871,Y -8.642,Z 104.656,A 1.708,B 90.000,C 0.000} C_DIS
LIN {X -289.869,Y -8.720,Z 104.549,A 1.723,B 90.000,C 0.000} C_DIS
LIN {X -289.867,Y -8.775,Z 104.354,A 1.734,B 90.000,C 0.000} C_DIS
LIN {X -289.864,Y -8.877,Z 104.282,A 1.754,B 90.000,C 0.000} C_DIS
LIN {X -289.863,Y -8.898,Z 104.192,A 1.758,B 90.000,C 0.000} C_DIS
LIN {X -289.862,Y -8.940,Z 104.070,A 1.767,B 90.000,C 0.000} C_DIS
LIN {X -289.856,Y -9.144,Z 103.848,A 1.807,B 90.000,C 0.000} C_DIS
LIN {X -289.854,Y -9.187,Z 103.726,A 1.815,B 90.000,C 0.000} C_DIS
LIN {X -289.854,Y -9.208,Z 103.635,A 1.820,B 90.000,C 0.000} C_DIS
LIN {X -289.851,Y -9.310,Z 103.560,A 1.840,B 90.000,C 0.000} C_DIS
LIN {X -289.850,Y -9.331,Z 103.469,A 1.844,B 90.000,C 0.000} C_DIS
LIN {X -289.848,Y -9.374,Z 103.348,A 1.852,B 90.000,C 0.000} C_DIS
LIN {X -289.842,Y -9.578,Z 103.125,A 1.893,B 90.000,C 0.000} C_DIS
LIN {X -289.840,Y -9.620,Z 103.004,A 1.901,B 90.000,C 0.000} C_DIS
LIN {X -289.840,Y -9.641,Z 102.913,A 1.905,B 90.000,C 0.000} C_DIS
LIN {X -289.836,Y -9.743,Z 102.832,A 1.925,B 90.000,C 0.000} C_DIS
LIN {X -289.835,Y -9.786,Z 102.628,A 1.934,B 90.000,C 0.000} C_DIS
LIN {X -289.831,Y -9.888,Z 102.548,A 1.954,B 90.000,C 0.000} C_DIS
LIN {X -289.831,Y -9.909,Z 102.457,A 1.958,B 90.000,C 0.000} C_DIS
LIN {X -289.829,Y -9.951,Z 102.336,A 1.966,B 90.000,C 0.000} C_DIS
LIN {X -289.822,Y -10.155,Z 102.113,A 2.007,B 90.000,C 0.000} C_DIS
LIN {X -289.821,Y -10.198,Z 101.992,A 2.015,B 90.000,C 0.000} C_DIS
LIN {X -289.820,Y -10.219,Z 101.901,A 2.019,B 90.000,C 0.000} C_DIS
LIN {X -289.816,Y -10.321,Z 101.825,A 2.040,B 90.000,C 0.000} C_DIS
LIN {X -289.816,Y -10.342,Z 101.735,A 2.044,B 90.000,C 0.000} C_DIS
LIN {X -289.814,Y -10.385,Z 101.613,A 2.052,B 90.000,C 0.000} C_DIS
LIN {X -289.807,Y -10.589,Z 101.391,A 2.092,B 90.000,C 0.000} C_DIS
LIN {X -289.805,Y -10.631,Z 101.269,A 2.101,B 90.000,C 0.000} C_DIS
LIN {X -289.804,Y -10.652,Z 101.178,A 2.105,B 90.000,C 0.000} C_DIS
LIN {X -289.801,Y -10.754,Z 101.103,A 2.125,B 90.000,C 0.000} C_DIS
LIN {X -289.800,Y -10.776,Z 101.012,A 2.129,B 90.000,C 0.000} C_DIS
LIN {X -289.798,Y -10.818,Z 100.891,A 2.138,B 90.000,C 0.000} C_DIS
LIN {X -289.790,Y -11.022,Z 100.668,A 2.178,B 90.000,C 0.000} C_DIS
LIN {X -289.789,Y -11.064,Z 100.547,A 2.187,B 90.000,C 0.000} C_DIS
LIN {X -289.788,Y -11.086,Z 100.456,A 2.191,B 90.000,C 0.000} C_DIS
LIN {X -289.784,Y -11.188,Z 100.380,A 2.211,B 90.000,C 0.000} C_DIS
LIN {X -289.783,Y -11.209,Z 100.289,A 2.215,B 90.000,C 0.000} C_DIS
LIN {X -289.782,Y -11.251,Z 100.168,A 2.223,B 90.000,C 0.000} C_DIS
LIN {X -289.774,Y -11.455,Z 99.945,A 2.264,B 90.000,C 0.000} C_DIS
LIN {X -289.772,Y -11.498,Z 99.824,A 2.272,B 90.000,C 0.000} C_DIS
LIN {X -289.771,Y -11.519,Z 99.733,A 2.276,B 90.000,C 0.000} C_DIS
LIN {X -289.767,Y -11.621,Z 99.658,A 2.297,B 90.000,C 0.000} C_DIS
LIN {X -289.766,Y -11.642,Z 99.567,A 2.301,B 90.000,C 0.000} C_DIS
LIN {X -289.765,Y -11.684,Z 99.445,A 2.309,B 90.000,C 0.000} C_DIS
LIN {X -289.756,Y -11.888,Z 99.223,A 2.349,B 90.000,C 0.000} C_DIS
LIN {X -289.754,Y -11.931,Z 99.101,A 2.358,B 90.000,C 0.000} C_DIS
LIN {X -289.754,Y -11.952,Z 99.010,A 2.362,B 90.000,C 0.000} C_DIS
LIN {X -289.749,Y -12.054,Z 98.935,A 2.382,B 90.000,C 0.000} C_DIS
LIN {X -289.748,Y -12.075,Z 98.844,A 2.386,B 90.000,C 0.000} C_DIS
LIN {X -289.747,Y -12.118,Z 98.723,A 2.395,B 90.000,C 0.000} C_DIS
LIN {X -289.738,Y -12.322,Z 98.500,A 2.435,B 90.000,C 0.000} C_DIS
LIN {X -289.736,Y -12.364,Z 98.379,A 2.444,B 90.000,C 0.000} C_DIS
LIN {X -289.735,Y -12.385,Z 98.288,A 2.448,B 90.000,C 0.000} C_DIS
LIN {X -289.731,Y -12.487,Z 98.212,A 2.468,B 90.000,C 0.000} C_DIS
LIN {X -289.730,Y -12.508,Z 98.121,A 2.472,B 90.000,C 0.000} C_DIS
LIN {X -289.728,Y -12.551,Z 98.000,A 2.480,B 90.000,C 0.000} C_DIS
LIN {X -289.719,Y -12.755,Z 97.777,A 2.521,B 90.000,C 0.000} C_DIS
LIN {X -289.718,Y -12.797,Z 97.656,A 2.529,B 90.000,C 0.000} C_DIS
LIN {X -289.717,Y -12.818,Z 97.565,A 2.533,B 90.000,C 0.000} C_DIS
LIN {X -289.712,Y -12.920,Z 97.490,A 2.554,B 90.000,C 0.000} C_DIS
LIN {X -289.711,Y -12.942,Z 97.399,A 2.558,B 90.000,C 0.000} C_DIS
LIN {X -289.709,Y -12.984,Z 97.277,A 2.566,B 90.000,C 0.000} C_DIS
LIN {X -289.700,Y -13.188,Z 97.055,A 2.606,B 90.000,C 0.000} C_DIS
LIN {X -289.698,Y -13.230,Z 96.933,A 2.615,B 90.000,C 0.000} C_DIS
LIN {X -289.697,Y -13.252,Z 96.843,A 2.619,B 90.000,C 0.000} C_DIS
LIN {X -289.692,Y -13.354,Z 96.762,A 2.639,B 90.000,C 0.000} C_DIS
LIN {X -289.690,Y -13.396,Z 96.558,A 2.648,B 90.000,C 0.000} C_DIS
LIN {X -289.686,Y -13.498,Z 96.478,A 2.668,B 90.000,C 0.000} C_DIS
LIN {X -289.685,Y -13.519,Z 96.387,A 2.672,B 90.000,C 0.000} C_DIS
LIN {X -289.683,Y -13.562,Z 96.266,A 2.680,B 90.000,C 0.000} C_DIS
LIN {X -289.673,Y -13.765,Z 96.043,A 2.721,B 90.000,C 0.000} C_DIS
LIN {X -289.671,Y -13.808,Z 95.922,A 2.729,B 90.000,C 0.000} C_DIS
LIN {X -289.670,Y -13.829,Z 95.831,A 2.733,B 90.000,C 0.000} C_DIS
LIN {X -289.665,Y -13.931,Z 95.755,A 2.753,B 90.000,C 0.000} C_DIS
LIN {X -289.664,Y -13.952,Z 95.664,A 2.758,B 90.000,C 0.000} C_DIS
LIN {X -289.662,Y -13.995,Z 95.543,A 2.766,B 90.000,C 0.000} C_DIS
LIN {X -289.652,Y -14.199,Z 95.320,A 2.806,B 90.000,C 0.000} C_DIS
LIN {X -289.650,Y -14.241,Z 95.199,A 2.815,B 90.000,C 0.000} C_DIS
LIN {X -289.649,Y -14.262,Z 95.108,A 2.819,B 90.000,C 0.000} C_DIS
LIN {X -289.644,Y -14.364,Z 95.033,A 2.839,B 90.000,C 0.000} C_DIS
LIN {X -289.643,Y -14.385,Z 94.942,A 2.843,B 90.000,C 0.000} C_DIS
LIN {X -289.641,Y -14.428,Z 94.820,A 2.852,B 90.000,C 0.000} C_DIS
LIN {X -289.631,Y -14.632,Z 94.598,A 2.892,B 90.000,C 0.000} C_DIS
LIN {X -289.629,Y -14.674,Z 94.476,A 2.900,B 90.000,C 0.000} C_DIS
LIN {X -289.627,Y -14.695,Z 94.386,A 2.905,B 90.000,C 0.000} C_DIS
LIN {X -289.622,Y -14.797,Z 94.310,A 2.925,B 90.000,C 0.000} C_DIS
LIN {X -289.621,Y -14.818,Z 94.219,A 2.929,B 90.000,C 0.000} C_DIS
LIN {X -289.619,Y -14.861,Z 94.098,A 2.937,B 90.000,C 0.000} C_DIS
LIN {X -289.608,Y -15.065,Z 93.875,A 2.978,B 90.000,C 0.000} C_DIS
LIN {X -289.606,Y -15.107,Z 93.754,A 2.986,B 90.000,C 0.000} C_DIS
LIN {X -289.605,Y -15.128,Z 93.663,A 2.990,B 90.000,C 0.000} C_DIS
LIN {X -289.600,Y -15.230,Z 93.587,A 3.010,B 90.000,C 0.000} C_DIS
LIN {X -289.599,Y -15.251,Z 93.497,A 3.015,B 90.000,C 0.000} C_DIS
LIN {X -289.596,Y -15.294,Z 93.375,A 3.023,B 90.000,C 0.000} C_DIS
LIN {X -289.586,Y -15.498,Z 93.152,A 3.063,B 90.000,C 0.000} C_DIS
LIN {X -289.583,Y -15.540,Z 93.031,A 3.072,B 90.000,C 0.000} C_DIS
LIN {X -289.582,Y -15.561,Z 92.940,A 3.076,B 90.000,C 0.000} C_DIS
LIN {X -289.577,Y -15.663,Z 92.865,A 3.096,B 90.000,C 0.000} C_DIS
LIN {X -289.576,Y -15.684,Z 92.774,A 3.100,B 90.000,C 0.000} C_DIS
LIN {X -289.573,Y -15.727,Z 92.652,A 3.109,B 90.000,C 0.000} C_DIS
LIN {X -289.562,Y -15.931,Z 92.430,A 3.149,B 90.000,C 0.000} C_DIS
LIN {X -289.560,Y -15.973,Z 92.308,A 3.157,B 90.000,C 0.000} C_DIS
LIN {X -289.559,Y -15.994,Z 92.218,A 3.162,B 90.000,C 0.000} C_DIS
LIN {X -289.553,Y -16.096,Z 92.142,A 3.182,B 90.000,C 0.000} C_DIS
LIN {X -289.552,Y -16.117,Z 92.051,A 3.186,B 90.000,C 0.000} C_DIS
LIN {X -289.549,Y -16.160,Z 91.930,A 3.194,B 90.000,C 0.000} C_DIS
LIN {X -289.538,Y -16.363,Z 91.707,A 3.235,B 90.000,C 0.000} C_DIS
LIN {X -289.536,Y -16.406,Z 91.586,A 3.243,B 90.000,C 0.000} C_DIS
LIN {X -289.534,Y -16.427,Z 91.495,A 3.247,B 90.000,C 0.000} C_DIS
LIN {X -289.529,Y -16.529,Z 91.419,A 3.267,B 90.000,C 0.000} C_DIS
LIN {X -289.527,Y -16.550,Z 91.329,A 3.272,B 90.000,C 0.000} C_DIS
LIN {X -289.525,Y -16.593,Z 91.207,A 3.280,B 90.000,C 0.000} C_DIS
LIN {X -289.513,Y -16.796,Z 90.985,A 3.320,B 90.000,C 0.000} C_DIS
LIN {X -289.511,Y -16.839,Z 90.863,A 3.329,B 90.000,C 0.000} C_DIS
LIN {X -289.509,Y -16.860,Z 90.772,A 3.333,B 90.000,C 0.000} C_DIS
LIN {X -289.504,Y -16.962,Z 90.697,A 3.353,B 90.000,C 0.000} C_DIS
LIN {X -289.502,Y -16.983,Z 90.606,A 3.357,B 90.000,C 0.000} C_DIS
LIN {X -289.500,Y -17.025,Z 90.485,A 3.366,B 90.000,C 0.000} C_DIS
LIN {X -289.488,Y -17.229,Z 90.262,A 3.406,B 90.000,C 0.000} C_DIS
LIN {X -289.485,Y -17.272,Z 90.140,A 3.414,B 90.000,C 0.000} C_DIS
LIN {X -289.484,Y -17.293,Z 90.050,A 3.419,B 90.000,C 0.000} C_DIS
LIN {X -289.478,Y -17.395,Z 89.969,A 3.439,B 90.000,C 0.000} C_DIS
LIN {X -289.475,Y -17.437,Z 89.765,A 3.447,B 90.000,C 0.000} C_DIS
LIN {X -289.469,Y -17.539,Z 89.685,A 3.467,B 90.000,C 0.000} C_DIS
LIN {X -289.468,Y -17.560,Z 89.594,A 3.472,B 90.000,C 0.000} C_DIS
LIN {X -289.465,Y -17.602,Z 89.473,A 3.480,B 90.000,C 0.000} C_DIS
LIN {X -289.453,Y -17.806,Z 89.250,A 3.520,B 90.000,C 0.000} C_DIS
LIN {X -289.450,Y -17.849,Z 89.129,A 3.529,B 90.000,C 0.000} C_DIS
LIN {X -289.449,Y -17.870,Z 89.038,A 3.533,B 90.000,C 0.000} C_DIS
LIN {X -289.443,Y -17.972,Z 88.962,A 3.553,B 90.000,C 0.000} C_DIS
LIN {X -289.441,Y -17.993,Z 88.872,A 3.557,B 90.000,C 0.000} C_DIS
LIN {X -289.439,Y -18.035,Z 88.750,A 3.566,B 90.000,C 0.000} C_DIS
LIN {X -289.426,Y -18.239,Z 88.528,A 3.606,B 90.000,C 0.000} C_DIS
LIN {X -289.423,Y -18.281,Z 88.406,A 3.614,B 90.000,C 0.000} C_DIS
LIN {X -289.422,Y -18.303,Z 88.315,A 3.618,B 90.000,C 0.000} C_DIS
LIN {X -289.415,Y -18.404,Z 88.240,A 3.639,B 90.000,C 0.000} C_DIS
LIN {X -289.414,Y -18.426,Z 88.149,A 3.643,B 90.000,C 0.000} C_DIS
LIN {X -289.411,Y -18.468,Z 88.028,A 3.651,B 90.000,C 0.000} C_DIS
LIN {X -289.398,Y -18.672,Z 87.805,A 3.692,B 90.000,C 0.000} C_DIS
LIN {X -289.396,Y -18.714,Z 87.684,A 3.700,B 90.000,C 0.000} C_DIS
LIN {X -289.394,Y -18.735,Z 87.593,A 3.704,B 90.000,C 0.000} C_DIS
LIN {X -289.388,Y -18.837,Z 87.517,A 3.724,B 90.000,C 0.000} C_DIS
LIN {X -289.386,Y -18.858,Z 87.426,A 3.728,B 90.000,C 0.000} C_DIS
LIN {X -289.383,Y -18.901,Z 87.305,A 3.737,B 90.000,C 0.000} C_DIS
LIN {X -289.370,Y -19.104,Z 87.082,A 3.777,B 90.000,C 0.000} C_DIS
LIN {X -289.367,Y -19.147,Z 86.961,A 3.786,B 90.000,C 0.000} C_DIS
LIN {X -289.366,Y -19.168,Z 86.870,A 3.790,B 90.000,C 0.000} C_DIS
LIN {X -289.359,Y -19.270,Z 86.795,A 3.810,B 90.000,C 0.000} C_DIS
LIN {X -289.358,Y -19.291,Z 86.704,A 3.814,B 90.000,C 0.000} C_DIS
LIN {X -289.355,Y -19.333,Z 86.582,A 3.823,B 90.000,C 0.000} C_DIS
LIN {X -289.341,Y -19.537,Z 86.360,A 3.863,B 90.000,C 0.000} C_DIS
LIN {X -289.338,Y -19.579,Z 86.238,A 3.871,B 90.000,C 0.000} C_DIS
LIN {X -289.337,Y -19.601,Z 86.147,A 3.875,B 90.000,C 0.000} C_DIS
LIN {X -289.330,Y -19.702,Z 86.072,A 3.896,B 90.000,C 0.000} C_DIS
LIN {X -289.329,Y -19.724,Z 85.981,A 3.900,B 90.000,C 0.000} C_DIS
LIN {X -289.326,Y -19.766,Z 85.860,A 3.908,B 90.000,C 0.000} C_DIS
LIN {X -289.312,Y -19.970,Z 85.637,A 3.949,B 90.000,C 0.000} C_DIS
LIN {X -289.309,Y -20.012,Z 85.516,A 3.957,B 90.000,C 0.000} C_DIS
LIN {X -289.307,Y -20.033,Z 85.425,A 3.961,B 90.000,C 0.000} C_DIS
LIN {X -289.300,Y -20.135,Z 85.349,A 3.981,B 90.000,C 0.000} C_DIS
LIN {X -289.299,Y -20.156,Z 85.258,A 3.985,B 90.000,C 0.000} C_DIS
LIN {X -289.296,Y -20.198,Z 85.137,A 3.994,B 90.000,C 0.000} C_DIS
LIN {X -289.281,Y -20.402,Z 84.914,A 4.034,B 90.000,C 0.000} C_DIS
LIN {X -289.278,Y -20.444,Z 84.793,A 4.043,B 90.000,C 0.000} C_DIS
LIN {X -289.277,Y -20.466,Z 84.702,A 4.047,B 90.000,C 0.000} C_DIS
LIN {X -289.270,Y -20.567,Z 84.627,A 4.067,B 90.000,C 0.000} C_DIS
LIN {X -289.268,Y -20.589,Z 84.536,A 4.071,B 90.000,C 0.000} C_DIS
LIN {X -289.265,Y -20.631,Z 84.414,A 4.080,B 90.000,C 0.000} C_DIS
LIN {X -289.251,Y -20.835,Z 84.192,A 4.120,B 90.000,C 0.000} C_DIS
LIN {X -289.248,Y -20.877,Z 84.070,A 4.128,B 90.000,C 0.000} C_DIS
LIN {X -289.246,Y -20.898,Z 83.980,A 4.132,B 90.000,C 0.000} C_DIS
LIN {X -289.239,Y -21.000,Z 83.899,A 4.153,B 90.000,C 0.000} C_DIS
LIN {X -289.236,Y -21.042,Z 83.695,A 4.161,B 90.000,C 0.000} C_DIS
LIN {X -289.228,Y -21.144,Z 83.615,A 4.181,B 90.000,C 0.000} C_DIS
LIN {X -289.227,Y -21.165,Z 83.524,A 4.185,B 90.000,C 0.000} C_DIS
LIN {X -289.224,Y -21.208,Z 83.403,A 4.194,B 90.000,C 0.000} C_DIS
LIN {X -289.209,Y -21.411,Z 83.180,A 4.234,B 90.000,C 0.000} C_DIS
LIN {X -289.205,Y -21.453,Z 83.059,A 4.242,B 90.000,C 0.000} C_DIS
LIN {X -289.204,Y -21.475,Z 82.968,A 4.247,B 90.000,C 0.000} C_DIS
LIN {X -289.196,Y -21.576,Z 82.892,A 4.267,B 90.000,C 0.000} C_DIS
LIN {X -289.195,Y -21.598,Z 82.801,A 4.271,B 90.000,C 0.000} C_DIS
LIN {X -289.191,Y -21.640,Z 82.680,A 4.279,B 90.000,C 0.000} C_DIS
LIN {X -289.176,Y -21.844,Z 82.457,A 4.320,B 90.000,C 0.000} C_DIS
LIN {X -289.173,Y -21.886,Z 82.336,A 4.328,B 90.000,C 0.000} C_DIS
LIN {X -289.171,Y -21.907,Z 82.245,A 4.332,B 90.000,C 0.000} C_DIS
LIN {X -289.164,Y -22.009,Z 82.170,A 4.353,B 90.000,C 0.000} C_DIS
LIN {X -289.162,Y -22.030,Z 82.079,A 4.357,B 90.000,C 0.000} C_DIS
LIN {X -289.159,Y -22.072,Z 81.957,A 4.365,B 90.000,C 0.000} C_DIS
LIN {X -289.143,Y -22.276,Z 81.735,A 4.405,B 90.000,C 0.000} C_DIS
LIN {X -289.140,Y -22.318,Z 81.613,A 4.414,B 90.000,C 0.000} C_DIS
LIN {X -289.138,Y -22.339,Z 81.523,A 4.418,B 90.000,C 0.000} C_DIS
LIN {X -289.130,Y -22.441,Z 81.447,A 4.438,B 90.000,C 0.000} C_DIS
LIN {X -289.129,Y -22.462,Z 81.356,A 4.442,B 90.000,C 0.000} C_DIS
LIN {X -289.125,Y -22.505,Z 81.235,A 4.451,B 90.000,C 0.000} C_DIS
LIN {X -289.110,Y -22.708,Z 81.012,A 4.491,B 90.000,C 0.000} C_DIS
LIN {X -289.106,Y -22.750,Z 80.891,A 4.499,B 90.000,C 0.000} C_DIS
LIN {X -289.105,Y -22.772,Z 80.800,A 4.504,B 90.000,C 0.000} C_DIS
LIN {X -289.097,Y -22.873,Z 80.724,A 4.524,B 90.000,C 0.000} C_DIS
LIN {X -289.095,Y -22.895,Z 80.634,A 4.528,B 90.000,C 0.000} C_DIS
LIN {X -289.092,Y -22.937,Z 80.512,A 4.536,B 90.000,C 0.000} C_DIS
LIN {X -289.075,Y -23.140,Z 80.289,A 4.577,B 90.000,C 0.000} C_DIS
LIN {X -289.072,Y -23.183,Z 80.168,A 4.585,B 90.000,C 0.000} C_DIS
LIN {X -289.070,Y -23.204,Z 80.077,A 4.589,B 90.000,C 0.000} C_DIS
LIN {X -289.062,Y -23.306,Z 80.002,A 4.609,B 90.000,C 0.000} C_DIS
LIN {X -289.060,Y -23.327,Z 79.911,A 4.614,B 90.000,C 0.000} C_DIS
LIN {X -289.057,Y -23.369,Z 79.789,A 4.622,B 90.000,C 0.000} C_DIS
LIN {X -289.040,Y -23.573,Z 79.567,A 4.662,B 90.000,C 0.000} C_DIS
LIN {X -289.037,Y -23.615,Z 79.445,A 4.671,B 90.000,C 0.000} C_DIS
LIN {X -289.035,Y -23.636,Z 79.355,A 4.675,B 90.000,C 0.000} C_DIS
LIN {X -289.027,Y -23.738,Z 79.279,A 4.695,B 90.000,C 0.000} C_DIS
LIN {X -289.025,Y -23.759,Z 79.188,A 4.699,B 90.000,C 0.000} C_DIS
LIN {X -289.022,Y -23.801,Z 79.067,A 4.708,B 90.000,C 0.000} C_DIS
LIN {X -289.005,Y -24.005,Z 78.844,A 4.748,B 90.000,C 0.000} C_DIS
LIN {X -289.001,Y -24.047,Z 78.723,A 4.756,B 90.000,C 0.000} C_DIS
LIN {X -289.000,Y -24.068,Z 78.632,A 4.761,B 90.000,C 0.000} C_DIS
LIN {X -288.991,Y -24.170,Z 78.556,A 4.781,B 90.000,C 0.000} C_DIS
LIN {X -288.989,Y -24.191,Z 78.466,A 4.785,B 90.000,C 0.000} C_DIS
LIN {X -288.986,Y -24.233,Z 78.344,A 4.793,B 90.000,C 0.000} C_DIS
LIN {X -288.969,Y -24.437,Z 78.122,A 4.834,B 90.000,C 0.000} C_DIS
LIN {X -288.965,Y -24.479,Z 78.000,A 4.842,B 90.000,C 0.000} C_DIS
LIN {X -288.963,Y -24.500,Z 77.909,A 4.846,B 90.000,C 0.000} C_DIS
LIN {X -288.955,Y -24.602,Z 77.834,A 4.866,B 90.000,C 0.000} C_DIS
LIN {X -288.953,Y -24.623,Z 77.743,A 4.871,B 90.000,C 0.000} C_DIS
LIN {X -288.949,Y -24.665,Z 77.622,A 4.879,B 90.000,C 0.000} C_DIS
LIN {X -288.932,Y -24.869,Z 77.399,A 4.919,B 90.000,C 0.000} C_DIS
LIN {X -288.928,Y -24.911,Z 77.277,A 4.928,B 90.000,C 0.000} C_DIS
LIN {X -288.926,Y -24.932,Z 77.187,A 4.932,B 90.000,C 0.000} C_DIS
LIN {X -288.917,Y -25.034,Z 77.106,A 4.952,B 90.000,C 0.000} C_DIS
LIN {X -288.914,Y -25.076,Z 76.902,A 4.961,B 90.000,C 0.000} C_DIS
LIN {X -288.905,Y -25.178,Z 76.822,A 4.981,B 90.000,C 0.000} C_DIS
LIN {X -288.903,Y -25.199,Z 76.731,A 4.985,B 90.000,C 0.000} C_DIS
LIN {X -288.899,Y -25.241,Z 76.610,A 4.993,B 90.000,C 0.000} C_DIS
LIN {X -288.882,Y -25.445,Z 76.387,A 5.034,B 90.000,C 0.000} C_DIS
LIN {X -288.878,Y -25.487,Z 76.266,A 5.042,B 90.000,C 0.000} C_DIS
LIN {X -288.876,Y -25.508,Z 76.175,A 5.046,B 90.000,C 0.000} C_DIS
LIN {X -288.867,Y -25.610,Z 76.099,A 5.066,B 90.000,C 0.000} C_DIS
LIN {X -288.865,Y -25.631,Z 76.009,A 5.071,B 90.000,C 0.000} C_DIS
LIN {X -288.861,Y -25.673,Z 75.887,A 5.079,B 90.000,C 0.000} C_DIS
LIN {X -288.843,Y -25.877,Z 75.665,A 5.119,B 90.000,C 0.000} C_DIS
LIN {X -288.839,Y -25.919,Z 75.543,A 5.128,B 90.000,C 0.000} C_DIS
LIN {X -288.838,Y -25.940,Z 75.452,A 5.132,B 90.000,C 0.000} C_DIS
LIN {X -288.828,Y -26.042,Z 75.377,A 5.152,B 90.000,C 0.000} C_DIS
LIN {X -288.826,Y -26.063,Z 75.286,A 5.156,B 90.000,C 0.000} C_DIS
LIN {X -288.823,Y -26.105,Z 75.165,A 5.165,B 90.000,C 0.000} C_DIS
LIN {X -288.804,Y -26.308,Z 74.942,A 5.205,B 90.000,C 0.000} C_DIS
LIN {X -288.800,Y -26.351,Z 74.821,A 5.213,B 90.000,C 0.000} C_DIS
LIN {X -288.798,Y -26.372,Z 74.730,A 5.218,B 90.000,C 0.000} C_DIS
LIN {X -288.789,Y -26.473,Z 74.654,A 5.238,B 90.000,C 0.000} C_DIS
LIN {X -288.787,Y -26.495,Z 74.563,A 5.242,B 90.000,C 0.000} C_DIS
LIN {X -288.783,Y -26.537,Z 74.442,A 5.250,B 90.000,C 0.000} C_DIS
LIN {X -288.765,Y -26.740,Z 74.219,A 5.291,B 90.000,C 0.000} C_DIS
LIN {X -288.761,Y -26.782,Z 74.098,A 5.299,B 90.000,C 0.000} C_DIS
LIN {X -288.759,Y -26.804,Z 74.007,A 5.303,B 90.000,C 0.000} C_DIS
LIN {X -288.749,Y -26.905,Z 73.932,A 5.323,B 90.000,C 0.000} C_DIS
LIN {X -288.747,Y -26.926,Z 73.841,A 5.328,B 90.000,C 0.000} C_DIS
LIN {X -288.743,Y -26.969,Z 73.719,A 5.336,B 90.000,C 0.000} C_DIS
LIN {X -288.724,Y -27.172,Z 73.497,A 5.376,B 90.000,C 0.000} C_DIS
LIN {X -288.720,Y -27.214,Z 73.375,A 5.385,B 90.000,C 0.000} C_DIS
LIN {X -288.718,Y -27.235,Z 73.284,A 5.389,B 90.000,C 0.000} C_DIS
LIN {X -288.709,Y -27.337,Z 73.209,A 5.409,B 90.000,C 0.000} C_DIS
LIN {X -288.707,Y -27.358,Z 73.118,A 5.413,B 90.000,C 0.000} C_DIS
LIN {X -288.703,Y -27.400,Z 72.997,A 5.422,B 90.000,C 0.000} C_DIS
LIN {X -288.683,Y -27.604,Z 72.774,A 5.462,B 90.000,C 0.000} C_DIS
LIN {X -288.679,Y -27.646,Z 72.653,A 5.470,B 90.000,C 0.000} C_DIS
LIN {X -288.677,Y -27.667,Z 72.562,A 5.475,B 90.000,C 0.000} C_DIS
LIN {X -288.667,Y -27.769,Z 72.486,A 5.495,B 90.000,C 0.000} C_DIS
LIN {X -288.665,Y -27.790,Z 72.395,A 5.499,B 90.000,C 0.000} C_DIS
LIN {X -288.661,Y -27.832,Z 72.274,A 5.507,B 90.000,C 0.000} C_DIS
LIN {X -288.642,Y -28.035,Z 72.051,A 5.548,B 90.000,C 0.000} C_DIS
LIN {X -288.638,Y -28.077,Z 71.930,A 5.556,B 90.000,C 0.000} C_DIS
LIN {X -288.636,Y -28.098,Z 71.839,A 5.560,B 90.000,C 0.000} C_DIS
LIN {X -288.626,Y -28.200,Z 71.764,A 5.580,B 90.000,C 0.000} C_DIS
LIN {X -288.624,Y -28.221,Z 71.673,A 5.585,B 90.000,C 0.000} C_DIS
LIN {X -288.619,Y -28.263,Z 71.551,A 5.593,B 90.000,C 0.000} C_DIS
LIN {X -288.599,Y -28.467,Z 71.329,A 5.633,B 90.000,C 0.000} C_DIS
LIN {X -288.595,Y -28.509,Z 71.207,A 5.642,B 90.000,C 0.000} C_DIS
LIN {X -288.593,Y -28.530,Z 71.116,A 5.646,B 90.000,C 0.000} C_DIS
LIN {X -288.583,Y -28.632,Z 71.036,A 5.666,B 90.000,C 0.000} C_DIS
LIN {X -288.579,Y -28.674,Z 70.832,A 5.674,B 90.000,C 0.000} C_DIS
LIN {X -288.569,Y -28.775,Z 70.752,A 5.695,B 90.000,C 0.000} C_DIS
LIN {X -288.567,Y -28.797,Z 70.661,A 5.699,B 90.000,C 0.000} C_DIS
LIN {X -288.563,Y -28.839,Z 70.540,A 5.707,B 90.000,C 0.000} C_DIS
LIN {X -288.542,Y -29.042,Z 70.317,A 5.747,B 90.000,C 0.000} C_DIS
LIN {X -288.538,Y -29.084,Z 70.196,A 5.756,B 90.000,C 0.000} C_DIS
LIN {X -288.536,Y -29.105,Z 70.105,A 5.760,B 90.000,C 0.000} C_DIS
LIN {X -288.525,Y -29.207,Z 70.029,A 5.780,B 90.000,C 0.000} C_DIS
LIN {X -288.523,Y -29.228,Z 69.938,A 5.784,B 90.000,C 0.000} C_DIS
LIN {X -288.519,Y -29.270,Z 69.817,A 5.793,B 90.000,C 0.000} C_DIS
LIN {X -288.498,Y -29.473,Z 69.594,A 5.833,B 90.000,C 0.000} C_DIS
LIN {X -288.494,Y -29.515,Z 69.473,A 5.842,B 90.000,C 0.000} C_DIS
LIN {X -288.492,Y -29.537,Z 69.382,A 5.846,B 90.000,C 0.000} C_DIS
LIN {X -288.482,Y -29.638,Z 69.307,A 5.866,B 90.000,C 0.000} C_DIS
LIN {X -288.479,Y -29.659,Z 69.216,A 5.870,B 90.000,C 0.000} C_DIS
LIN {X -288.475,Y -29.701,Z 69.094,A 5.878,B 90.000,C 0.000} C_DIS
LIN {X -288.454,Y -29.905,Z 68.872,A 5.919,B 90.000,C 0.000} C_DIS
LIN {X -288.450,Y -29.947,Z 68.750,A 5.927,B 90.000,C 0.000} C_DIS
LIN {X -288.447,Y -29.968,Z 68.660,A 5.931,B 90.000,C 0.000} C_DIS
LIN {X -288.437,Y -30.069,Z 68.584,A 5.952,B 90.000,C 0.000} C_DIS
LIN {X -288.435,Y -30.091,Z 68.493,A 5.956,B 90.000,C 0.000} C_DIS
LIN {X -288.430,Y -30.133,Z 68.372,A 5.964,B 90.000,C 0.000} C_DIS
LIN {X -288.409,Y -30.336,Z 68.149,A 6.004,B 90.000,C 0.000} C_DIS
LIN {X -288.405,Y -30.378,Z 68.028,A 6.013,B 90.000,C 0.000} C_DIS
LIN {X -288.402,Y -30.399,Z 67.937,A 6.017,B 90.000,C 0.000} C_DIS
LIN {X -288.392,Y -30.501,Z 67.861,A 6.037,B 90.000,C 0.000} C_DIS
LIN {X -288.389,Y -30.522,Z 67.771,A 6.041,B 90.000,C 0.000} C_DIS
LIN {X -288.385,Y -30.564,Z 67.649,A 6.050,B 90.000,C 0.000} C_DIS
LIN {X -288.363,Y -30.767,Z 67.426,A 6.090,B 90.000,C 0.000} C_DIS
LIN {X -288.359,Y -30.809,Z 67.305,A 6.099,B 90.000,C 0.000} C_DIS
LIN {X -288.357,Y -30.830,Z 67.214,A 6.103,B 90.000,C 0.000} C_DIS
LIN {X -288.346,Y -30.932,Z 67.139,A 6.123,B 90.000,C 0.000} C_DIS
LIN {X -288.343,Y -30.953,Z 67.048,A 6.127,B 90.000,C 0.000} C_DIS
LIN {X -288.339,Y -30.995,Z 66.926,A 6.135,B 90.000,C 0.000} C_DIS
LIN {X -288.317,Y -31.198,Z 66.704,A 6.176,B 90.000,C 0.000} C_DIS
LIN {X -288.312,Y -31.240,Z 66.582,A 6.184,B 90.000,C 0.000} C_DIS
LIN {X -288.310,Y -31.261,Z 66.492,A 6.188,B 90.000,C 0.000} C_DIS
LIN {X -288.299,Y -31.363,Z 66.416,A 6.209,B 90.000,C 0.000} C_DIS
LIN {X -288.297,Y -31.384,Z 66.325,A 6.213,B 90.000,C 0.000} C_DIS
LIN {X -288.292,Y -31.426,Z 66.204,A 6.221,B 90.000,C 0.000} C_DIS
LIN {X -288.270,Y -31.629,Z 65.981,A 6.261,B 90.000,C 0.000} C_DIS
LIN {X -288.265,Y -31.671,Z 65.860,A 6.270,B 90.000,C 0.000} C_DIS
LIN {X -288.263,Y -31.692,Z 65.769,A 6.274,B 90.000,C 0.000} C_DIS
LIN {X -288.252,Y -31.794,Z 65.689,A 6.294,B 90.000,C 0.000} C_DIS
LIN {X -288.247,Y -31.836,Z 65.485,A 6.303,B 90.000,C 0.000} C_DIS
LIN {X -288.236,Y -31.938,Z 65.404,A 6.323,B 90.000,C 0.000} C_DIS
LIN {X -288.234,Y -31.959,Z 65.314,A 6.327,B 90.000,C 0.000} C_DIS
LIN {X -288.229,Y -32.001,Z 65.192,A 6.335,B 90.000,C 0.000} C_DIS
LIN {X -288.206,Y -32.204,Z 64.969,A 6.376,B 90.000,C 0.000} C_DIS
LIN {X -288.202,Y -32.246,Z 64.848,A 6.384,B 90.000,C 0.000} C_DIS
LIN {X -288.199,Y -32.267,Z 64.757,A 6.388,B 90.000,C 0.000} C_DIS
LIN {X -288.188,Y -32.368,Z 64.682,A 6.408,B 90.000,C 0.000} C_DIS
LIN {X -288.186,Y -32.390,Z 64.591,A 6.413,B 90.000,C 0.000} C_DIS
LIN {X -288.181,Y -32.432,Z 64.470,A 6.421,B 90.000,C 0.000} C_DIS
LIN {X -288.158,Y -32.635,Z 64.247,A 6.461,B 90.000,C 0.000} C_DIS
LIN {X -288.153,Y -32.677,Z 64.125,A 6.470,B 90.000,C 0.000} C_DIS
LIN {X -288.151,Y -32.698,Z 64.035,A 6.474,B 90.000,C 0.000} C_DIS
LIN {X -288.139,Y -32.799,Z 63.959,A 6.494,B 90.000,C 0.000} C_DIS
LIN {X -288.137,Y -32.820,Z 63.868,A 6.498,B 90.000,C 0.000} C_DIS
LIN {X -288.132,Y -32.863,Z 63.747,A 6.507,B 90.000,C 0.000} C_DIS
LIN {X -288.109,Y -33.065,Z 63.524,A 6.547,B 90.000,C 0.000} C_DIS
LIN {X -288.104,Y -33.108,Z 63.403,A 6.555,B 90.000,C 0.000} C_DIS
LIN {X -288.102,Y -33.129,Z 63.312,A 6.560,B 90.000,C 0.000} C_DIS
LIN {X -288.090,Y -33.230,Z 63.236,A 6.580,B 90.000,C 0.000} C_DIS
LIN {X -288.087,Y -33.251,Z 63.146,A 6.584,B 90.000,C 0.000} C_DIS
LIN {X -288.083,Y -33.293,Z 63.024,A 6.592,B 90.000,C 0.000} C_DIS
LIN {X -288.059,Y -33.496,Z 62.802,A 6.633,B 90.000,C 0.000} C_DIS
LIN {X -288.054,Y -33.538,Z 62.680,A 6.641,B 90.000,C 0.000} C_DIS
LIN {X -288.052,Y -33.559,Z 62.589,A 6.645,B 90.000,C 0.000} C_DIS
LIN {X -288.040,Y -33.661,Z 62.514,A 6.665,B 90.000,C 0.000} C_DIS
LIN {X -288.037,Y -33.682,Z 62.423,A 6.670,B 90.000,C 0.000} C_DIS
LIN {X -288.032,Y -33.724,Z 62.302,A 6.678,B 90.000,C 0.000} C_DIS
LIN {X -288.009,Y -33.927,Z 62.079,A 6.718,B 90.000,C 0.000} C_DIS
LIN {X -288.004,Y -33.969,Z 61.957,A 6.727,B 90.000,C 0.000} C_DIS
LIN {X -288.001,Y -33.990,Z 61.867,A 6.731,B 90.000,C 0.000} C_DIS
LIN {X -287.989,Y -34.091,Z 61.791,A 6.751,B 90.000,C 0.000} C_DIS
LIN {X -287.987,Y -34.112,Z 61.700,A 6.755,B 90.000,C 0.000} C_DIS
LIN {X -287.982,Y -34.155,Z 61.579,A 6.764,B 90.000,C 0.000} C_DIS
LIN {X -287.958,Y -34.357,Z 61.356,A 6.804,B 90.000,C 0.000} C_DIS
LIN {X -287.953,Y -34.399,Z 61.235,A 6.812,B 90.000,C 0.000} C_DIS
LIN {X -287.950,Y -34.421,Z 61.144,A 6.817,B 90.000,C 0.000} C_DIS
LIN {X -287.938,Y -34.522,Z 61.069,A 6.837,B 90.000,C 0.000} C_DIS
LIN {X -287.935,Y -34.543,Z 60.978,A 6.841,B 90.000,C 0.000} C_DIS
LIN {X -287.930,Y -34.585,Z 60.856,A 6.849,B 90.000,C 0.000} C_DIS
LIN {X -287.906,Y -34.788,Z 60.634,A 6.890,B 90.000,C 0.000} C_DIS
LIN {X -287.901,Y -34.830,Z 60.512,A 6.898,B 90.000,C 0.000} C_DIS
LIN {X -287.898,Y -34.851,Z 60.421,A 6.902,B 90.000,C 0.000} C_DIS
LIN {X -287.886,Y -34.952,Z 60.346,A 6.922,B 90.000,C 0.000} C_DIS
LIN {X -287.883,Y -34.973,Z 60.255,A 6.927,B 90.000,C 0.000} C_DIS
LIN {X -287.878,Y -35.016,Z 60.134,A 6.935,B 90.000,C 0.000} C_DIS
LIN {X -287.854,Y -35.218,Z 59.911,A 6.975,B 90.000,C 0.000} C_DIS
LIN {X -287.848,Y -35.260,Z 59.790,A 6.984,B 90.000,C 0.000} C_DIS
LIN {X -287.846,Y -35.281,Z 59.699,A 6.988,B 90.000,C 0.000} C_DIS
LIN {X -287.833,Y -35.383,Z 59.623,A 7.008,B 90.000,C 0.000} C_DIS
LIN {X -287.831,Y -35.404,Z 59.532,A 7.012,B 90.000,C 0.000} C_DIS
LIN {X -287.826,Y -35.446,Z 59.411,A 7.021,B 90.000,C 0.000} C_DIS
LIN {X -287.801,Y -35.649,Z 59.188,A 7.061,B 90.000,C 0.000} C_DIS
LIN {X -287.795,Y -35.691,Z 59.067,A 7.069,B 90.000,C 0.000} C_DIS
LIN {X -287.793,Y -35.712,Z 58.976,A 7.074,B 90.000,C 0.000} C_DIS
LIN {X -287.780,Y -35.813,Z 58.901,A 7.094,B 90.000,C 0.000} C_DIS
LIN {X -287.778,Y -35.834,Z 58.810,A 7.098,B 90.000,C 0.000} C_DIS
LIN {X -287.772,Y -35.876,Z 58.688,A 7.106,B 90.000,C 0.000} C_DIS
LIN {X -287.747,Y -36.079,Z 58.466,A 7.147,B 90.000,C 0.000} C_DIS
LIN {X -287.742,Y -36.121,Z 58.344,A 7.155,B 90.000,C 0.000} C_DIS
LIN {X -287.739,Y -36.142,Z 58.253,A 7.159,B 90.000,C 0.000} C_DIS
LIN {X -287.726,Y -36.243,Z 58.173,A 7.179,B 90.000,C 0.000} C_DIS
LIN {X -287.721,Y -36.285,Z 57.969,A 7.188,B 90.000,C 0.000} C_DIS
LIN {X -287.708,Y -36.387,Z 57.889,A 7.208,B 90.000,C 0.000} C_DIS
LIN {X -287.706,Y -36.408,Z 57.798,A 7.212,B 90.000,C 0.000} C_DIS
LIN {X -287.700,Y -36.450,Z 57.677,A 7.221,B 90.000,C 0.000} C_DIS
LIN {X -287.674,Y -36.652,Z 57.454,A 7.261,B 90.000,C 0.000} C_DIS
LIN {X -287.669,Y -36.694,Z 57.333,A 7.269,B 90.000,C 0.000} C_DIS
LIN {X -287.666,Y -36.716,Z 57.242,A 7.273,B 90.000,C 0.000} C_DIS
LIN {X -287.653,Y -36.817,Z 57.166,A 7.294,B 90.000,C 0.000} C_DIS
LIN {X -287.651,Y -36.838,Z 57.075,A 7.298,B 90.000,C 0.000} C_DIS
LIN {X -287.645,Y -36.880,Z 56.954,A 7.306,B 90.000,C 0.000} C_DIS
LIN {X -287.619,Y -37.082,Z 56.731,A 7.347,B 90.000,C 0.000} C_DIS
LIN {X -287.614,Y -37.125,Z 56.610,A 7.355,B 90.000,C 0.000} C_DIS
LIN {X -287.611,Y -37.146,Z 56.519,A 7.359,B 90.000,C 0.000} C_DIS
LIN {X -287.598,Y -37.247,Z 56.444,A 7.379,B 90.000,C 0.000} C_DIS
LIN {X -287.595,Y -37.268,Z 56.353,A 7.383,B 90.000,C 0.000} C_DIS
LIN {X -287.590,Y -37.310,Z 56.231,A 7.392,B 90.000,C 0.000} C_DIS
LIN {X -287.564,Y -37.512,Z 56.009,A 7.432,B 90.000,C 0.000} C_DIS
LIN {X -287.558,Y -37.555,Z 55.887,A 7.441,B 90.000,C 0.000} C_DIS
LIN {X -287.555,Y -37.576,Z 55.797,A 7.445,B 90.000,C 0.000} C_DIS
LIN {X -287.542,Y -37.677,Z 55.721,A 7.465,B 90.000,C 0.000} C_DIS
LIN {X -287.539,Y -37.698,Z 55.630,A 7.469,B 90.000,C 0.000} C_DIS
LIN {X -287.534,Y -37.740,Z 55.509,A 7.478,B 90.000,C 0.000} C_DIS
LIN {X -287.507,Y -37.942,Z 55.286,A 7.518,B 90.000,C 0.000} C_DIS
LIN {X -287.502,Y -37.984,Z 55.165,A 7.526,B 90.000,C 0.000} C_DIS
LIN {X -287.499,Y -38.005,Z 55.074,A 7.530,B 90.000,C 0.000} C_DIS
LIN {X -287.485,Y -38.107,Z 54.998,A 7.551,B 90.000,C 0.000} C_DIS
LIN {X -287.483,Y -38.128,Z 54.908,A 7.555,B 90.000,C 0.000} C_DIS
LIN {X -287.477,Y -38.170,Z 54.786,A 7.563,B 90.000,C 0.000} C_DIS
LIN {X -287.450,Y -38.372,Z 54.563,A 7.604,B 90.000,C 0.000} C_DIS
LIN {X -287.445,Y -38.414,Z 54.442,A 7.612,B 90.000,C 0.000} C_DIS
LIN {X -287.442,Y -38.435,Z 54.351,A 7.616,B 90.000,C 0.000} C_DIS
LIN {X -287.428,Y -38.536,Z 54.276,A 7.636,B 90.000,C 0.000} C_DIS
LIN {X -287.425,Y -38.557,Z 54.185,A 7.640,B 90.000,C 0.000} C_DIS
LIN {X -287.420,Y -38.600,Z 54.063,A 7.649,B 90.000,C 0.000} C_DIS
LIN {X -287.392,Y -38.802,Z 53.841,A 7.689,B 90.000,C 0.000} C_DIS
LIN {X -287.387,Y -38.844,Z 53.719,A 7.698,B 90.000,C 0.000} C_DIS
LIN {X -287.384,Y -38.865,Z 53.629,A 7.702,B 90.000,C 0.000} C_DIS
LIN {X -287.370,Y -38.966,Z 53.553,A 7.722,B 90.000,C 0.000} C_DIS
LIN {X -287.367,Y -38.987,Z 53.462,A 7.726,B 90.000,C 0.000} C_DIS
LIN {X -287.362,Y -39.029,Z 53.341,A 7.735,B 90.000,C 0.000} C_DIS
LIN {X -287.334,Y -39.231,Z 53.118,A 7.775,B 90.000,C 0.000} C_DIS
LIN {X -287.328,Y -39.274,Z 52.997,A 7.783,B 90.000,C 0.000} C_DIS
LIN {X -287.325,Y -39.295,Z 52.906,A 7.787,B 90.000,C 0.000} C_DIS
LIN {X -287.312,Y -39.396,Z 52.830,A 7.808,B 90.000,C 0.000} C_DIS
LIN {X -287.309,Y -39.417,Z 52.740,A 7.812,B 90.000,C 0.000} C_DIS
LIN {X -287.303,Y -39.459,Z 52.618,A 7.820,B 90.000,C 0.000} C_DIS
LIN {X -287.275,Y -39.661,Z 52.396,A 7.861,B 90.000,C 0.000} C_DIS
LIN {X -287.269,Y -39.703,Z 52.274,A 7.869,B 90.000,C 0.000} C_DIS
LIN {X -287.266,Y -39.724,Z 52.183,A 7.873,B 90.000,C 0.000} C_DIS
LIN {X -287.252,Y -39.825,Z 52.103,A 7.893,B 90.000,C 0.000} C_DIS
LIN {X -287.247,Y -39.867,Z 51.899,A 7.902,B 90.000,C 0.000} C_DIS
LIN {X -287.233,Y -39.968,Z 51.819,A 7.922,B 90.000,C 0.000} C_DIS
LIN {X -287.230,Y -39.989,Z 51.728,A 7.926,B 90.000,C 0.000} C_DIS
LIN {X -287.224,Y -40.031,Z 51.606,A 7.934,B 90.000,C 0.000} C_DIS
LIN {X -287.195,Y -40.234,Z 51.384,A 7.975,B 90.000,C 0.000} C_DIS
LIN {X -287.190,Y -40.276,Z 51.262,A 7.983,B 90.000,C 0.000} C_DIS
LIN {X -287.187,Y -40.297,Z 51.172,A 7.987,B 90.000,C 0.000} C_DIS
LIN {X -287.172,Y -40.398,Z 51.096,A 8.008,B 90.000,C 0.000} C_DIS
LIN {X -287.169,Y -40.419,Z 51.005,A 8.012,B 90.000,C 0.000} C_DIS
LIN {X -287.164,Y -40.461,Z 50.884,A 8.020,B 90.000,C 0.000} C_DIS
LIN {X -287.135,Y -40.663,Z 50.661,A 8.060,B 90.000,C 0.000} C_DIS
LIN {X -287.129,Y -40.705,Z 50.540,A 8.069,B 90.000,C 0.000} C_DIS
LIN {X -287.126,Y -40.726,Z 50.449,A 8.073,B 90.000,C 0.000} C_DIS
LIN {X -287.112,Y -40.827,Z 50.369,A 8.093,B 90.000,C 0.000} C_DIS
LIN {X -287.106,Y -40.869,Z 50.165,A 8.102,B 90.000,C 0.000} C_DIS
LIN {X -287.091,Y -40.970,Z 50.080,A 8.122,B 90.000,C 0.000} C_DIS
LIN {X -287.085,Y -41.012,Z 49.876,A 8.130,B 90.000,C 0.000} C_DIS
LIN {X -287.071,Y -41.113,Z 49.791,A 8.150,B 90.000,C 0.000} C_DIS
LIN {X -287.065,Y -41.155,Z 49.586,A 8.159,B 90.000,C 0.000} C_DIS
LIN {X -287.058,Y -41.206,Z 49.544,A 8.169,B 90.000,C 0.000} C_DIS
LIN {X -287.050,Y -41.256,Z 49.480,A 8.179,B 90.000,C 0.000} C_DIS
LIN {X -287.044,Y -41.298,Z 49.174,A 8.187,B 90.000,C 0.000} C_DIS
LIN {X -287.030,Y -41.399,Z 49.047,A 8.207,B 90.000,C 0.000} C_DIS
LIN {X -287.024,Y -41.441,Z 48.741,A 8.216,B 90.000,C 0.000} C_DIS
LIN {X -287.016,Y -41.492,Z 48.677,A 8.226,B 90.000,C 0.000} C_DIS
LIN {X -287.009,Y -41.542,Z 48.592,A 8.236,B 90.000,C 0.000} C_DIS
LIN {X -287.003,Y -41.584,Z 48.184,A 8.244,B 90.000,C 0.000} C_DIS
LIN {X -286.996,Y -41.635,Z 48.099,A 8.254,B 90.000,C 0.000} C_DIS
LIN {X -286.988,Y -41.687,Z 47.846,A 8.265,B 90.000,C 0.000} C_DIS
LIN {X -286.988,Y -41.687,Z 46.473,A 8.265,B 90.000,C 0.000} C_DIS
LIN {X -286.996,Y -41.635,Z 46.220,A 8.254,B 90.000,C 0.000} C_DIS
LIN {X -287.003,Y -41.584,Z 46.135,A 8.244,B 90.000,C 0.000} C_DIS
LIN {X -287.009,Y -41.542,Z 45.727,A 8.236,B 90.000,C 0.000} C_DIS
LIN {X -287.016,Y -41.492,Z 45.642,A 8.226,B 90.000,C 0.000} C_DIS
LIN {X -287.024,Y -41.441,Z 45.578,A 8.216,B 90.000,C 0.000} C_DIS
LIN {X -287.030,Y -41.399,Z 45.272,A 8.207,B 90.000,C 0.000} C_DIS
LIN {X -287.037,Y -41.349,Z 45.208,A 8.197,B 90.000,C 0.000} C_DIS
LIN {X -287.044,Y -41.298,Z 45.170,A 8.187,B 90.000,C 0.000} C_DIS
LIN {X -287.047,Y -41.277,Z 45.080,A 8.183,B 90.000,C 0.000} C_DIS
LIN {X -287.053,Y -41.235,Z 44.958,A 8.175,B 90.000,C 0.000} C_DIS
LIN {X -287.068,Y -41.134,Z 44.847,A 8.154,B 90.000,C 0.000} C_DIS
LIN {X -287.112,Y -40.825,Z 44.410,A 8.093,B 90.000,C 0.000} C_DIS
LIN {X -287.221,Y -40.052,Z 43.639,A 7.938,B 90.000,C 0.000} C_DIS
LIN {X -287.254,Y -39.812,Z 43.474,A 7.891,B 90.000,C 0.000} C_DIS
LIN {X -287.265,Y -39.735,Z 43.453,A 7.875,B 90.000,C 0.000} C_DIS
LIN {X -287.269,Y -39.703,Z 43.402,A 7.869,B 90.000,C 0.000} C_DIS
LIN {X -287.275,Y -39.661,Z 43.351,A 7.861,B 90.000,C 0.000} C_DIS
LIN {X -287.303,Y -39.459,Z 43.308,A 7.820,B 90.000,C 0.000} C_DIS
LIN {X -287.315,Y -39.375,Z 43.206,A 7.803,B 90.000,C 0.000} C_DIS
LIN {X -287.342,Y -39.172,Z 43.164,A 7.763,B 90.000,C 0.000} C_DIS
LIN {X -287.354,Y -39.088,Z 43.061,A 7.746,B 90.000,C 0.000} C_DIS
LIN {X -287.381,Y -38.886,Z 43.019,A 7.706,B 90.000,C 0.000} C_DIS
LIN {X -287.387,Y -38.844,Z 42.968,A 7.698,B 90.000,C 0.000} C_DIS
LIN {X -287.395,Y -38.781,Z 42.917,A 7.685,B 90.000,C 0.000} C_DIS
LIN {X -287.436,Y -38.477,Z 42.874,A 7.625,B 90.000,C 0.000} C_DIS
LIN {X -287.445,Y -38.414,Z 42.823,A 7.612,B 90.000,C 0.000} C_DIS
LIN {X -287.456,Y -38.330,Z 42.772,A 7.595,B 90.000,C 0.000} C_DIS
LIN {X -287.509,Y -37.925,Z 42.730,A 7.514,B 90.000,C 0.000} C_DIS
LIN {X -287.521,Y -37.841,Z 42.679,A 7.498,B 90.000,C 0.000} C_DIS
LIN {X -287.556,Y -37.572,Z 42.626,A 7.444,B 90.000,C 0.000} C_DIS
LIN {X -287.744,Y -36.103,Z 42.626,A 7.151,B 90.000,C 0.000} C_DIS
LIN {X -287.778,Y -35.834,Z 42.679,A 7.098,B 90.000,C 0.000} C_DIS
LIN {X -287.785,Y -35.771,Z 42.730,A 7.085,B 90.000,C 0.000} C_DIS
LIN {X -287.823,Y -35.467,Z 42.772,A 7.025,B 90.000,C 0.000} C_DIS
LIN {X -287.839,Y -35.341,Z 42.874,A 7.000,B 90.000,C 0.000} C_DIS
LIN {X -287.876,Y -35.037,Z 42.917,A 6.939,B 90.000,C 0.000} C_DIS
LIN {X -287.883,Y -34.973,Z 42.968,A 6.927,B 90.000,C 0.000} C_DIS
LIN {X -287.889,Y -34.931,Z 43.019,A 6.918,B 90.000,C 0.000} C_DIS
LIN {X -287.913,Y -34.729,Z 43.061,A 6.878,B 90.000,C 0.000} C_DIS
LIN {X -287.923,Y -34.644,Z 43.164,A 6.861,B 90.000,C 0.000} C_DIS
LIN {X -287.948,Y -34.442,Z 43.206,A 6.821,B 90.000,C 0.000} C_DIS
LIN {X -287.957,Y -34.362,Z 43.308,A 6.805,B 90.000,C 0.000} C_DIS
LIN {X -287.968,Y -34.272,Z 43.329,A 6.787,B 90.000,C 0.000} C_DIS
LIN {X -287.982,Y -34.151,Z 43.372,A 6.763,B 90.000,C 0.000} C_DIS
LIN {X -287.995,Y -34.041,Z 43.474,A 6.741,B 90.000,C 0.000} C_DIS
LIN {X -288.051,Y -33.566,Z 43.830,A 6.647,B 90.000,C 0.000} C_DIS
LIN {X -288.162,Y -32.600,Z 44.803,A 6.454,B 90.000,C 0.000} C_DIS
LIN {X -288.202,Y -32.246,Z 45.280,A 6.384,B 90.000,C 0.000} C_DIS
LIN {X -288.213,Y -32.144,Z 45.392,A 6.364,B 90.000,C 0.000} C_DIS
LIN {X -288.218,Y -32.102,Z 45.513,A 6.356,B 90.000,C 0.000} C_DIS
LIN {X -288.220,Y -32.081,Z 45.604,A 6.351,B 90.000,C 0.000} C_DIS
LIN {X -288.231,Y -31.980,Z 45.679,A 6.331,B 90.000,C 0.000} C_DIS
LIN {X -288.234,Y -31.959,Z 45.770,A 6.327,B 90.000,C 0.000} C_DIS
LIN {X -288.238,Y -31.916,Z 45.892,A 6.319,B 90.000,C 0.000} C_DIS
LIN {X -288.261,Y -31.711,Z 46.134,A 6.278,B 90.000,C 0.000} C_DIS
LIN {X -288.268,Y -31.650,Z 46.450,A 6.266,B 90.000,C 0.000} C_DIS
LIN {X -288.273,Y -31.599,Z 46.509,A 6.256,B 90.000,C 0.000} C_DIS
LIN {X -288.279,Y -31.549,Z 46.551,A 6.245,B 90.000,C 0.000} C_DIS
LIN {X -288.283,Y -31.507,Z 46.755,A 6.237,B 90.000,C 0.000} C_DIS
LIN {X -288.295,Y -31.405,Z 46.840,A 6.217,B 90.000,C 0.000} C_DIS
LIN {X -288.299,Y -31.363,Z 47.045,A 6.209,B 90.000,C 0.000} C_DIS
LIN {X -288.305,Y -31.312,Z 47.087,A 6.198,B 90.000,C 0.000} C_DIS
LIN {X -288.310,Y -31.261,Z 47.151,A 6.188,B 90.000,C 0.000} C_DIS
LIN {X -288.315,Y -31.219,Z 47.457,A 6.180,B 90.000,C 0.000} C_DIS
LIN {X -288.326,Y -31.118,Z 47.584,A 6.160,B 90.000,C 0.000} C_DIS
LIN {X -288.330,Y -31.075,Z 47.890,A 6.151,B 90.000,C 0.000} C_DIS
LIN {X -288.336,Y -31.025,Z 47.954,A 6.141,B 90.000,C 0.000} C_DIS
LIN {X -288.341,Y -30.974,Z 47.997,A 6.131,B 90.000,C 0.000} C_DIS
LIN {X -288.346,Y -30.932,Z 48.201,A 6.123,B 90.000,C 0.000} C_DIS
LIN {X -288.351,Y -30.881,Z 48.243,A 6.113,B 90.000,C 0.000} C_DIS
LIN {X -288.357,Y -30.830,Z 48.307,A 6.103,B 90.000,C 0.000} C_DIS
LIN {X -288.361,Y -30.788,Z 48.613,A 6.094,B 90.000,C 0.000} C_DIS
LIN {X -288.366,Y -30.737,Z 48.677,A 6.084,B 90.000,C 0.000} C_DIS
LIN {X -288.372,Y -30.687,Z 48.719,A 6.074,B 90.000,C 0.000} C_DIS
LIN {X -288.376,Y -30.644,Z 48.923,A 6.066,B 90.000,C 0.000} C_DIS
LIN {X -288.382,Y -30.594,Z 48.966,A 6.056,B 90.000,C 0.000} C_DIS
LIN {X -288.387,Y -30.543,Z 49.030,A 6.046,B 90.000,C 0.000} C_DIS
LIN {X -288.392,Y -30.501,Z 49.336,A 6.037,B 90.000,C 0.000} C_DIS
LIN {X -288.397,Y -30.450,Z 49.399,A 6.027,B 90.000,C 0.000} C_DIS
LIN {X -288.402,Y -30.399,Z 49.442,A 6.017,B 90.000,C 0.000} C_DIS
LIN {X -288.407,Y -30.357,Z 49.646,A 6.009,B 90.000,C 0.000} C_DIS
LIN {X -288.412,Y -30.306,Z 49.689,A 5.999,B 90.000,C 0.000} C_DIS
LIN {X -288.417,Y -30.255,Z 49.752,A 5.989,B 90.000,C 0.000} C_DIS
LIN {X -288.422,Y -30.213,Z 50.058,A 5.980,B 90.000,C 0.000} C_DIS
LIN {X -288.427,Y -30.162,Z 50.122,A 5.970,B 90.000,C 0.000} C_DIS
LIN {X -288.432,Y -30.112,Z 50.165,A 5.960,B 90.000,C 0.000} C_DIS
LIN {X -288.437,Y -30.069,Z 50.369,A 5.952,B 90.000,C 0.000} C_DIS
LIN {X -288.442,Y -30.019,Z 50.411,A 5.941,B 90.000,C 0.000} C_DIS
LIN {X -288.447,Y -29.968,Z 50.475,A 5.931,B 90.000,C 0.000} C_DIS
LIN {X -288.452,Y -29.926,Z 50.781,A 5.923,B 90.000,C 0.000} C_DIS
LIN {X -288.457,Y -29.875,Z 50.845,A 5.913,B 90.000,C 0.000} C_DIS
LIN {X -288.462,Y -29.824,Z 50.887,A 5.903,B 90.000,C 0.000} C_DIS
LIN {X -288.467,Y -29.782,Z 51.091,A 5.894,B 90.000,C 0.000} C_DIS
LIN {X -288.472,Y -29.731,Z 51.134,A 5.884,B 90.000,C 0.000} C_DIS
LIN {X -288.477,Y -29.680,Z 51.197,A 5.874,B 90.000,C 0.000} C_DIS
LIN {X -288.482,Y -29.638,Z 51.504,A 5.866,B 90.000,C 0.000} C_DIS
LIN {X -288.487,Y -29.587,Z 51.567,A 5.856,B 90.000,C 0.000} C_DIS
LIN {X -288.492,Y -29.537,Z 51.610,A 5.846,B 90.000,C 0.000} C_DIS
LIN {X -288.496,Y -29.494,Z 51.814,A 5.837,B 90.000,C 0.000} C_DIS
LIN {X -288.501,Y -29.444,Z 51.856,A 5.827,B 90.000,C 0.000} C_DIS
LIN {X -288.507,Y -29.393,Z 51.920,A 5.817,B 90.000,C 0.000} C_DIS
LIN {X -288.511,Y -29.351,Z 52.226,A 5.809,B 90.000,C 0.000} C_DIS
LIN {X -288.516,Y -29.300,Z 52.290,A 5.799,B 90.000,C 0.000} C_DIS
LIN {X -288.521,Y -29.249,Z 52.332,A 5.789,B 90.000,C 0.000} C_DIS
LIN {X -288.525,Y -29.207,Z 52.537,A 5.780,B 90.000,C 0.000} C_DIS
LIN {X -288.531,Y -29.156,Z 52.579,A 5.770,B 90.000,C 0.000} C_DIS
LIN {X -288.536,Y -29.105,Z 52.643,A 5.760,B 90.000,C 0.000} C_DIS
LIN {X -288.540,Y -29.063,Z 52.949,A 5.752,B 90.000,C 0.000} C_DIS
LIN {X -288.545,Y -29.012,Z 53.013,A 5.742,B 90.000,C 0.000} C_DIS
LIN {X -288.550,Y -28.961,Z 53.055,A 5.732,B 90.000,C 0.000} C_DIS
LIN {X -288.554,Y -28.919,Z 53.259,A 5.723,B 90.000,C 0.000} C_DIS
LIN {X -288.560,Y -28.868,Z 53.302,A 5.713,B 90.000,C 0.000} C_DIS
LIN {X -288.565,Y -28.818,Z 53.365,A 5.703,B 90.000,C 0.000} C_DIS
LIN {X -288.569,Y -28.775,Z 53.672,A 5.695,B 90.000,C 0.000} C_DIS
LIN {X -288.574,Y -28.725,Z 53.735,A 5.684,B 90.000,C 0.000} C_DIS
LIN {X -288.579,Y -28.674,Z 53.778,A 5.674,B 90.000,C 0.000} C_DIS
LIN {X -288.583,Y -28.632,Z 53.982,A 5.666,B 90.000,C 0.000} C_DIS
LIN {X -288.588,Y -28.581,Z 54.024,A 5.656,B 90.000,C 0.000} C_DIS
LIN {X -288.593,Y -28.530,Z 54.088,A 5.646,B 90.000,C 0.000} C_DIS
LIN {X -288.597,Y -28.488,Z 54.394,A 5.637,B 90.000,C 0.000} C_DIS
LIN {X -288.602,Y -28.437,Z 54.458,A 5.627,B 90.000,C 0.000} C_DIS
LIN {X -288.607,Y -28.386,Z 54.500,A 5.617,B 90.000,C 0.000} C_DIS
LIN {X -288.612,Y -28.344,Z 54.705,A 5.609,B 90.000,C 0.000} C_DIS
LIN {X -288.617,Y -28.293,Z 54.747,A 5.599,B 90.000,C 0.000} C_DIS
LIN {X -288.622,Y -28.242,Z 54.811,A 5.589,B 90.000,C 0.000} C_DIS
LIN {X -288.626,Y -28.200,Z 55.117,A 5.580,B 90.000,C 0.000} C_DIS
LIN {X -288.631,Y -28.149,Z 55.181,A 5.570,B 90.000,C 0.000} C_DIS
LIN {X -288.636,Y -28.098,Z 55.223,A 5.560,B 90.000,C 0.000} C_DIS
LIN {X -288.640,Y -28.056,Z 55.427,A 5.552,B 90.000,C 0.000} C_DIS
LIN {X -288.645,Y -28.005,Z 55.470,A 5.542,B 90.000,C 0.000} C_DIS
LIN {X -288.650,Y -27.955,Z 55.533,A 5.532,B 90.000,C 0.000} C_DIS
LIN {X -288.654,Y -27.912,Z 55.840,A 5.523,B 90.000,C 0.000} C_DIS
LIN {X -288.659,Y -27.862,Z 55.903,A 5.513,B 90.000,C 0.000} C_DIS
LIN {X -288.663,Y -27.811,Z 55.946,A 5.503,B 90.000,C 0.000} C_DIS
LIN {X -288.667,Y -27.768,Z 56.150,A 5.495,B 90.000,C 0.000} C_DIS
LIN {X -288.672,Y -27.718,Z 56.192,A 5.485,B 90.000,C 0.000} C_DIS
LIN {X -288.677,Y -27.667,Z 56.256,A 5.475,B 90.000,C 0.000} C_DIS
LIN {X -288.681,Y -27.625,Z 56.562,A 5.466,B 90.000,C 0.000} C_DIS
LIN {X -288.686,Y -27.574,Z 56.626,A 5.456,B 90.000,C 0.000} C_DIS
LIN {X -288.691,Y -27.523,Z 56.668,A 5.446,B 90.000,C 0.000} C_DIS
LIN {X -288.695,Y -27.481,Z 56.872,A 5.438,B 90.000,C 0.000} C_DIS
LIN {X -288.700,Y -27.430,Z 56.915,A 5.427,B 90.000,C 0.000} C_DIS
LIN {X -288.705,Y -27.379,Z 56.979,A 5.417,B 90.000,C 0.000} C_DIS
LIN {X -288.709,Y -27.337,Z 57.285,A 5.409,B 90.000,C 0.000} C_DIS
LIN {X -288.713,Y -27.286,Z 57.349,A 5.399,B 90.000,C 0.000} C_DIS
LIN {X -288.718,Y -27.235,Z 57.391,A 5.389,B 90.000,C 0.000} C_DIS
LIN {X -288.722,Y -27.193,Z 57.595,A 5.380,B 90.000,C 0.000} C_DIS
LIN {X -288.727,Y -27.142,Z 57.638,A 5.370,B 90.000,C 0.000} C_DIS
LIN {X -288.732,Y -27.091,Z 57.701,A 5.360,B 90.000,C 0.000} C_DIS
LIN {X -288.736,Y -27.049,Z 58.007,A 5.352,B 90.000,C 0.000} C_DIS
LIN {X -288.741,Y -26.998,Z 58.071,A 5.342,B 90.000,C 0.000} C_DIS
LIN {X -288.745,Y -26.947,Z 58.114,A 5.332,B 90.000,C 0.000} C_DIS
LIN {X -288.749,Y -26.905,Z 58.318,A 5.323,B 90.000,C 0.000} C_DIS
LIN {X -288.754,Y -26.854,Z 58.360,A 5.313,B 90.000,C 0.000} C_DIS
